// ---- DUTs/IO/Boxes/EL1808_78E8D3DD.TcDUT
{attribute 'GeneratedUsingTerminal: EL1808-0000-0016'}
{attribute addProperty BoxType "EL1808-0000-0016"}
{attribute addProperty Description "EL1808 8Ch. Dig. Input 24V, 3ms"}
{attribute addProperty Physics "KK"}
{attribute addProperty Id "Channel_1AT %I*Channel_830843C11Channel_2AT %I*Channel_830843C11Channel_3AT %I*Channel_830843C11Channel_4AT %I*Channel_830843C11Channel_5AT %I*Channel_830843C11Channel_6AT %I*Channel_830843C11Channel_7AT %I*Channel_830843C11Channel_8AT %I*Channel_830843C11WcStateAT %I*WcState_9091E0EB2InfoDataAT %I*InfoData_6F19DB2B2"}
{attribute addProperty CRC "2028524509"}
{attribute addProperty Size "12"}
TYPE EL1808_78E8D3DD EXTENDS EtcSlaveTerminalBase_947E5A46 :
STRUCT
	{attribute addProperty Name "Channel_1"}
	Channel_1 : Channel_830843C1;
	{attribute addProperty Name "Channel_2"}
	Channel_2 : Channel_830843C1;
	{attribute addProperty Name "Channel_3"}
	Channel_3 : Channel_830843C1;
	{attribute addProperty Name "Channel_4"}
	Channel_4 : Channel_830843C1;
	{attribute addProperty Name "Channel_5"}
	Channel_5 : Channel_830843C1;
	{attribute addProperty Name "Channel_6"}
	Channel_6 : Channel_830843C1;
	{attribute addProperty Name "Channel_7"}
	Channel_7 : Channel_830843C1;
	{attribute addProperty Name "Channel_8"}
	Channel_8 : Channel_830843C1;
	{attribute addProperty Name "WcState"}
	WcState : WcState_9091E0EB;
	{attribute addProperty Name "InfoData"}
	InfoData : InfoData_6F19DB2B;
END_STRUCT
END_TYPE

// ---- DUTs/IO/Boxes/EL1809_32157CFD.TcDUT
{attribute 'GeneratedUsingTerminal: EL1809-0000-0016'}
{attribute addProperty BoxType "EL1809-0000-0016"}
{attribute addProperty Description "EL1809 16Ch. Dig. Input 24V, 3ms"}
{attribute addProperty Physics "KK"}
{attribute addProperty Id "Channel_1AT %I*Channel_830843C11Channel_2AT %I*Channel_830843C11Channel_3AT %I*Channel_830843C11Channel_4AT %I*Channel_830843C11Channel_5AT %I*Channel_830843C11Channel_6AT %I*Channel_830843C11Channel_7AT %I*Channel_830843C11Channel_8AT %I*Channel_830843C11Channel_9AT %I*Channel_830843C11Channel_10AT %I*Channel_830843C11Channel_11AT %I*Channel_830843C11Channel_12AT %I*Channel_830843C11Channel_13AT %I*Channel_830843C11Channel_14AT %I*Channel_830843C11Channel_15AT %I*Channel_830843C11Channel_16AT %I*Channel_830843C11WcStateAT %I*WcState_9091E0EB2InfoDataAT %I*InfoData_6F19DB2B2"}
{attribute addProperty CRC "840269053"}
{attribute addProperty Size "20"}
TYPE EL1809_32157CFD EXTENDS EtcSlaveTerminalBase_947E5A46 :
STRUCT
	{attribute addProperty Name "Channel_1"}
	Channel_1 : Channel_830843C1;
	{attribute addProperty Name "Channel_2"}
	Channel_2 : Channel_830843C1;
	{attribute addProperty Name "Channel_3"}
	Channel_3 : Channel_830843C1;
	{attribute addProperty Name "Channel_4"}
	Channel_4 : Channel_830843C1;
	{attribute addProperty Name "Channel_5"}
	Channel_5 : Channel_830843C1;
	{attribute addProperty Name "Channel_6"}
	Channel_6 : Channel_830843C1;
	{attribute addProperty Name "Channel_7"}
	Channel_7 : Channel_830843C1;
	{attribute addProperty Name "Channel_8"}
	Channel_8 : Channel_830843C1;
	{attribute addProperty Name "Channel_9"}
	Channel_9 : Channel_830843C1;
	{attribute addProperty Name "Channel_10"}
	Channel_10 : Channel_830843C1;
	{attribute addProperty Name "Channel_11"}
	Channel_11 : Channel_830843C1;
	{attribute addProperty Name "Channel_12"}
	Channel_12 : Channel_830843C1;
	{attribute addProperty Name "Channel_13"}
	Channel_13 : Channel_830843C1;
	{attribute addProperty Name "Channel_14"}
	Channel_14 : Channel_830843C1;
	{attribute addProperty Name "Channel_15"}
	Channel_15 : Channel_830843C1;
	{attribute addProperty Name "Channel_16"}
	Channel_16 : Channel_830843C1;
	{attribute addProperty Name "WcState"}
	WcState : WcState_9091E0EB;
	{attribute addProperty Name "InfoData"}
	InfoData : InfoData_6F19DB2B;
END_STRUCT
END_TYPE

// ---- DUTs/IO/Boxes/EL1814_D135F8DB.TcDUT
{attribute 'GeneratedUsingTerminal: EL1814-0000-0016'}
{attribute addProperty BoxType "EL1814-0000-0016"}
{attribute addProperty Description "EL1814 4Ch. Dig. Input 24V, 10µs"}
{attribute addProperty Physics "KK"}
{attribute addProperty Id "Channel_1AT %I*Channel_830843C11Channel_2AT %I*Channel_830843C11Channel_3AT %I*Channel_830843C11Channel_4AT %I*Channel_830843C11WcStateAT %I*WcState_9091E0EB2InfoDataAT %I*InfoData_6F19DB2B2"}
{attribute addProperty CRC "3509975259"}
{attribute addProperty Size "8"}
TYPE EL1814_D135F8DB EXTENDS EtcSlaveTerminalBase_947E5A46 :
STRUCT
	{attribute addProperty Name "Channel_1"}
	Channel_1 : Channel_830843C1;
	{attribute addProperty Name "Channel_2"}
	Channel_2 : Channel_830843C1;
	{attribute addProperty Name "Channel_3"}
	Channel_3 : Channel_830843C1;
	{attribute addProperty Name "Channel_4"}
	Channel_4 : Channel_830843C1;
	{attribute addProperty Name "WcState"}
	WcState : WcState_9091E0EB;
	{attribute addProperty Name "InfoData"}
	InfoData : InfoData_6F19DB2B;
END_STRUCT
END_TYPE

// ---- DUTs/IO/Boxes/EL1819_32157CFD.TcDUT
{attribute 'GeneratedUsingTerminal: EL1819-0000-0016'}
{attribute addProperty BoxType "EL1819-0000-0016"}
{attribute addProperty Description "EL1819 16Ch. Dig. Input 24V, 10µs"}
{attribute addProperty Physics "KK"}
{attribute addProperty Id "Channel_1AT %I*Channel_830843C11Channel_2AT %I*Channel_830843C11Channel_3AT %I*Channel_830843C11Channel_4AT %I*Channel_830843C11Channel_5AT %I*Channel_830843C11Channel_6AT %I*Channel_830843C11Channel_7AT %I*Channel_830843C11Channel_8AT %I*Channel_830843C11Channel_9AT %I*Channel_830843C11Channel_10AT %I*Channel_830843C11Channel_11AT %I*Channel_830843C11Channel_12AT %I*Channel_830843C11Channel_13AT %I*Channel_830843C11Channel_14AT %I*Channel_830843C11Channel_15AT %I*Channel_830843C11Channel_16AT %I*Channel_830843C11WcStateAT %I*WcState_9091E0EB2InfoDataAT %I*InfoData_6F19DB2B2"}
{attribute addProperty CRC "840269053"}
{attribute addProperty Size "20"}
TYPE EL1819_32157CFD EXTENDS EtcSlaveTerminalBase_947E5A46 :
STRUCT
	{attribute addProperty Name "Channel_1"}
	Channel_1 : Channel_830843C1;
	{attribute addProperty Name "Channel_2"}
	Channel_2 : Channel_830843C1;
	{attribute addProperty Name "Channel_3"}
	Channel_3 : Channel_830843C1;
	{attribute addProperty Name "Channel_4"}
	Channel_4 : Channel_830843C1;
	{attribute addProperty Name "Channel_5"}
	Channel_5 : Channel_830843C1;
	{attribute addProperty Name "Channel_6"}
	Channel_6 : Channel_830843C1;
	{attribute addProperty Name "Channel_7"}
	Channel_7 : Channel_830843C1;
	{attribute addProperty Name "Channel_8"}
	Channel_8 : Channel_830843C1;
	{attribute addProperty Name "Channel_9"}
	Channel_9 : Channel_830843C1;
	{attribute addProperty Name "Channel_10"}
	Channel_10 : Channel_830843C1;
	{attribute addProperty Name "Channel_11"}
	Channel_11 : Channel_830843C1;
	{attribute addProperty Name "Channel_12"}
	Channel_12 : Channel_830843C1;
	{attribute addProperty Name "Channel_13"}
	Channel_13 : Channel_830843C1;
	{attribute addProperty Name "Channel_14"}
	Channel_14 : Channel_830843C1;
	{attribute addProperty Name "Channel_15"}
	Channel_15 : Channel_830843C1;
	{attribute addProperty Name "Channel_16"}
	Channel_16 : Channel_830843C1;
	{attribute addProperty Name "WcState"}
	WcState : WcState_9091E0EB;
	{attribute addProperty Name "InfoData"}
	InfoData : InfoData_6F19DB2B;
END_STRUCT
END_TYPE

// ---- DUTs/IO/Boxes/EL1852_7699BCF6.TcDUT
{attribute 'GeneratedUsingTerminal: EL1852-0000-0016'}
{attribute addProperty BoxType "EL1852-0000-0016"}
{attribute addProperty Description "EL1852 8Ch. Dig. Input 24V, 3ms, 8Ch. Dig. Output 24V, 0.5A"}
{attribute addProperty Physics "KK"}
{attribute addProperty Id "Channel_1AT %I*Channel_830843C11Channel_2AT %I*Channel_830843C11Channel_3AT %I*Channel_830843C11Channel_4AT %I*Channel_830843C11Channel_5AT %I*Channel_830843C11Channel_6AT %I*Channel_830843C11Channel_7AT %I*Channel_830843C11Channel_8AT %I*Channel_830843C11Channel_9AT %Q*Channel_42CA91F71Channel_10AT %Q*Channel_42CA91F71Channel_11AT %Q*Channel_42CA91F71Channel_12AT %Q*Channel_42CA91F71Channel_13AT %Q*Channel_42CA91F71Channel_14AT %Q*Channel_42CA91F71Channel_15AT %Q*Channel_42CA91F71Channel_16AT %Q*Channel_42CA91F71WcStateAT %I*WcState_9091E0EB2InfoDataAT %I*InfoData_6F19DB2B2"}
{attribute addProperty CRC "1989786870"}
{attribute addProperty Size "20"}
TYPE EL1852_7699BCF6 EXTENDS EtcSlaveTerminalBase_947E5A46 :
STRUCT
	{attribute addProperty Name "Channel_1"}
	Channel_1 : Channel_830843C1;
	{attribute addProperty Name "Channel_2"}
	Channel_2 : Channel_830843C1;
	{attribute addProperty Name "Channel_3"}
	Channel_3 : Channel_830843C1;
	{attribute addProperty Name "Channel_4"}
	Channel_4 : Channel_830843C1;
	{attribute addProperty Name "Channel_5"}
	Channel_5 : Channel_830843C1;
	{attribute addProperty Name "Channel_6"}
	Channel_6 : Channel_830843C1;
	{attribute addProperty Name "Channel_7"}
	Channel_7 : Channel_830843C1;
	{attribute addProperty Name "Channel_8"}
	Channel_8 : Channel_830843C1;
	{attribute addProperty Name "Channel_9"}
	Channel_9 : Channel_42CA91F7;
	{attribute addProperty Name "Channel_10"}
	Channel_10 : Channel_42CA91F7;
	{attribute addProperty Name "Channel_11"}
	Channel_11 : Channel_42CA91F7;
	{attribute addProperty Name "Channel_12"}
	Channel_12 : Channel_42CA91F7;
	{attribute addProperty Name "Channel_13"}
	Channel_13 : Channel_42CA91F7;
	{attribute addProperty Name "Channel_14"}
	Channel_14 : Channel_42CA91F7;
	{attribute addProperty Name "Channel_15"}
	Channel_15 : Channel_42CA91F7;
	{attribute addProperty Name "Channel_16"}
	Channel_16 : Channel_42CA91F7;
	{attribute addProperty Name "WcState"}
	WcState : WcState_9091E0EB;
	{attribute addProperty Name "InfoData"}
	InfoData : InfoData_6F19DB2B;
END_STRUCT
END_TYPE

// ---- DUTs/IO/Boxes/EL1859_7699BCF6.TcDUT
{attribute 'GeneratedUsingTerminal: EL1859-0000-0016'}
{attribute addProperty BoxType "EL1859-0000-0016"}
{attribute addProperty Description "EL1859 8Ch. Dig. Input 24V, 3ms, 8Ch. Dig. Output 24V, 0.5A"}
{attribute addProperty Physics "KK"}
{attribute addProperty Id "Channel_1AT %I*Channel_830843C11Channel_2AT %I*Channel_830843C11Channel_3AT %I*Channel_830843C11Channel_4AT %I*Channel_830843C11Channel_5AT %I*Channel_830843C11Channel_6AT %I*Channel_830843C11Channel_7AT %I*Channel_830843C11Channel_8AT %I*Channel_830843C11Channel_9AT %Q*Channel_42CA91F71Channel_10AT %Q*Channel_42CA91F71Channel_11AT %Q*Channel_42CA91F71Channel_12AT %Q*Channel_42CA91F71Channel_13AT %Q*Channel_42CA91F71Channel_14AT %Q*Channel_42CA91F71Channel_15AT %Q*Channel_42CA91F71Channel_16AT %Q*Channel_42CA91F71WcStateAT %I*WcState_9091E0EB2InfoDataAT %I*InfoData_6F19DB2B2"}
{attribute addProperty CRC "1989786870"}
{attribute addProperty Size "20"}
TYPE EL1859_7699BCF6 EXTENDS EtcSlaveTerminalBase_947E5A46 :
STRUCT
	{attribute addProperty Name "Channel_1"}
	Channel_1 : Channel_830843C1;
	{attribute addProperty Name "Channel_2"}
	Channel_2 : Channel_830843C1;
	{attribute addProperty Name "Channel_3"}
	Channel_3 : Channel_830843C1;
	{attribute addProperty Name "Channel_4"}
	Channel_4 : Channel_830843C1;
	{attribute addProperty Name "Channel_5"}
	Channel_5 : Channel_830843C1;
	{attribute addProperty Name "Channel_6"}
	Channel_6 : Channel_830843C1;
	{attribute addProperty Name "Channel_7"}
	Channel_7 : Channel_830843C1;
	{attribute addProperty Name "Channel_8"}
	Channel_8 : Channel_830843C1;
	{attribute addProperty Name "Channel_9"}
	Channel_9 : Channel_42CA91F7;
	{attribute addProperty Name "Channel_10"}
	Channel_10 : Channel_42CA91F7;
	{attribute addProperty Name "Channel_11"}
	Channel_11 : Channel_42CA91F7;
	{attribute addProperty Name "Channel_12"}
	Channel_12 : Channel_42CA91F7;
	{attribute addProperty Name "Channel_13"}
	Channel_13 : Channel_42CA91F7;
	{attribute addProperty Name "Channel_14"}
	Channel_14 : Channel_42CA91F7;
	{attribute addProperty Name "Channel_15"}
	Channel_15 : Channel_42CA91F7;
	{attribute addProperty Name "Channel_16"}
	Channel_16 : Channel_42CA91F7;
	{attribute addProperty Name "WcState"}
	WcState : WcState_9091E0EB;
	{attribute addProperty Name "InfoData"}
	InfoData : InfoData_6F19DB2B;
END_STRUCT
END_TYPE

// ---- DUTs/IO/Boxes/EL1862_32157CFD.TcDUT
{attribute 'GeneratedUsingTerminal: EL1862-0000-0016'}
{attribute addProperty BoxType "EL1862-0000-0016"}
{attribute addProperty Description "EL1862 16Ch. Dig. Input 24V, 3ms"}
{attribute addProperty Physics "KK"}
{attribute addProperty Id "Channel_1AT %I*Channel_830843C11Channel_2AT %I*Channel_830843C11Channel_3AT %I*Channel_830843C11Channel_4AT %I*Channel_830843C11Channel_5AT %I*Channel_830843C11Channel_6AT %I*Channel_830843C11Channel_7AT %I*Channel_830843C11Channel_8AT %I*Channel_830843C11Channel_9AT %I*Channel_830843C11Channel_10AT %I*Channel_830843C11Channel_11AT %I*Channel_830843C11Channel_12AT %I*Channel_830843C11Channel_13AT %I*Channel_830843C11Channel_14AT %I*Channel_830843C11Channel_15AT %I*Channel_830843C11Channel_16AT %I*Channel_830843C11WcStateAT %I*WcState_9091E0EB2InfoDataAT %I*InfoData_6F19DB2B2"}
{attribute addProperty CRC "840269053"}
{attribute addProperty Size "20"}
TYPE EL1862_32157CFD EXTENDS EtcSlaveTerminalBase_947E5A46 :
STRUCT
	{attribute addProperty Name "Channel_1"}
	Channel_1 : Channel_830843C1;
	{attribute addProperty Name "Channel_2"}
	Channel_2 : Channel_830843C1;
	{attribute addProperty Name "Channel_3"}
	Channel_3 : Channel_830843C1;
	{attribute addProperty Name "Channel_4"}
	Channel_4 : Channel_830843C1;
	{attribute addProperty Name "Channel_5"}
	Channel_5 : Channel_830843C1;
	{attribute addProperty Name "Channel_6"}
	Channel_6 : Channel_830843C1;
	{attribute addProperty Name "Channel_7"}
	Channel_7 : Channel_830843C1;
	{attribute addProperty Name "Channel_8"}
	Channel_8 : Channel_830843C1;
	{attribute addProperty Name "Channel_9"}
	Channel_9 : Channel_830843C1;
	{attribute addProperty Name "Channel_10"}
	Channel_10 : Channel_830843C1;
	{attribute addProperty Name "Channel_11"}
	Channel_11 : Channel_830843C1;
	{attribute addProperty Name "Channel_12"}
	Channel_12 : Channel_830843C1;
	{attribute addProperty Name "Channel_13"}
	Channel_13 : Channel_830843C1;
	{attribute addProperty Name "Channel_14"}
	Channel_14 : Channel_830843C1;
	{attribute addProperty Name "Channel_15"}
	Channel_15 : Channel_830843C1;
	{attribute addProperty Name "Channel_16"}
	Channel_16 : Channel_830843C1;
	{attribute addProperty Name "WcState"}
	WcState : WcState_9091E0EB;
	{attribute addProperty Name "InfoData"}
	InfoData : InfoData_6F19DB2B;
END_STRUCT
END_TYPE

// ---- DUTs/IO/Boxes/EL1872_32157CFD.TcDUT
{attribute 'GeneratedUsingTerminal: EL1872-0000-0016'}
{attribute addProperty BoxType "EL1872-0000-0016"}
{attribute addProperty Description "EL1872 16Ch. Dig. Input 24V, 10µs"}
{attribute addProperty Physics "KK"}
{attribute addProperty Id "Channel_1AT %I*Channel_830843C11Channel_2AT %I*Channel_830843C11Channel_3AT %I*Channel_830843C11Channel_4AT %I*Channel_830843C11Channel_5AT %I*Channel_830843C11Channel_6AT %I*Channel_830843C11Channel_7AT %I*Channel_830843C11Channel_8AT %I*Channel_830843C11Channel_9AT %I*Channel_830843C11Channel_10AT %I*Channel_830843C11Channel_11AT %I*Channel_830843C11Channel_12AT %I*Channel_830843C11Channel_13AT %I*Channel_830843C11Channel_14AT %I*Channel_830843C11Channel_15AT %I*Channel_830843C11Channel_16AT %I*Channel_830843C11WcStateAT %I*WcState_9091E0EB2InfoDataAT %I*InfoData_6F19DB2B2"}
{attribute addProperty CRC "840269053"}
{attribute addProperty Size "20"}
TYPE EL1872_32157CFD EXTENDS EtcSlaveTerminalBase_947E5A46 :
STRUCT
	{attribute addProperty Name "Channel_1"}
	Channel_1 : Channel_830843C1;
	{attribute addProperty Name "Channel_2"}
	Channel_2 : Channel_830843C1;
	{attribute addProperty Name "Channel_3"}
	Channel_3 : Channel_830843C1;
	{attribute addProperty Name "Channel_4"}
	Channel_4 : Channel_830843C1;
	{attribute addProperty Name "Channel_5"}
	Channel_5 : Channel_830843C1;
	{attribute addProperty Name "Channel_6"}
	Channel_6 : Channel_830843C1;
	{attribute addProperty Name "Channel_7"}
	Channel_7 : Channel_830843C1;
	{attribute addProperty Name "Channel_8"}
	Channel_8 : Channel_830843C1;
	{attribute addProperty Name "Channel_9"}
	Channel_9 : Channel_830843C1;
	{attribute addProperty Name "Channel_10"}
	Channel_10 : Channel_830843C1;
	{attribute addProperty Name "Channel_11"}
	Channel_11 : Channel_830843C1;
	{attribute addProperty Name "Channel_12"}
	Channel_12 : Channel_830843C1;
	{attribute addProperty Name "Channel_13"}
	Channel_13 : Channel_830843C1;
	{attribute addProperty Name "Channel_14"}
	Channel_14 : Channel_830843C1;
	{attribute addProperty Name "Channel_15"}
	Channel_15 : Channel_830843C1;
	{attribute addProperty Name "Channel_16"}
	Channel_16 : Channel_830843C1;
	{attribute addProperty Name "WcState"}
	WcState : WcState_9091E0EB;
	{attribute addProperty Name "InfoData"}
	InfoData : InfoData_6F19DB2B;
END_STRUCT
END_TYPE

// ---- DUTs/IO/Boxes/EL1889_32157CFD.TcDUT
{attribute 'GeneratedUsingTerminal: EL1889-0000-0016'}
{attribute addProperty BoxType "EL1889-0000-0016"}
{attribute addProperty Description "EL1889 16Ch. Dig. Input 24V, 3ms, negative"}
{attribute addProperty Physics "KK"}
{attribute addProperty Id "Channel_1AT %I*Channel_830843C11Channel_2AT %I*Channel_830843C11Channel_3AT %I*Channel_830843C11Channel_4AT %I*Channel_830843C11Channel_5AT %I*Channel_830843C11Channel_6AT %I*Channel_830843C11Channel_7AT %I*Channel_830843C11Channel_8AT %I*Channel_830843C11Channel_9AT %I*Channel_830843C11Channel_10AT %I*Channel_830843C11Channel_11AT %I*Channel_830843C11Channel_12AT %I*Channel_830843C11Channel_13AT %I*Channel_830843C11Channel_14AT %I*Channel_830843C11Channel_15AT %I*Channel_830843C11Channel_16AT %I*Channel_830843C11WcStateAT %I*WcState_9091E0EB2InfoDataAT %I*InfoData_6F19DB2B2"}
{attribute addProperty CRC "840269053"}
{attribute addProperty Size "20"}
TYPE EL1889_32157CFD EXTENDS EtcSlaveTerminalBase_947E5A46 :
STRUCT
	{attribute addProperty Name "Channel_1"}
	Channel_1 : Channel_830843C1;
	{attribute addProperty Name "Channel_2"}
	Channel_2 : Channel_830843C1;
	{attribute addProperty Name "Channel_3"}
	Channel_3 : Channel_830843C1;
	{attribute addProperty Name "Channel_4"}
	Channel_4 : Channel_830843C1;
	{attribute addProperty Name "Channel_5"}
	Channel_5 : Channel_830843C1;
	{attribute addProperty Name "Channel_6"}
	Channel_6 : Channel_830843C1;
	{attribute addProperty Name "Channel_7"}
	Channel_7 : Channel_830843C1;
	{attribute addProperty Name "Channel_8"}
	Channel_8 : Channel_830843C1;
	{attribute addProperty Name "Channel_9"}
	Channel_9 : Channel_830843C1;
	{attribute addProperty Name "Channel_10"}
	Channel_10 : Channel_830843C1;
	{attribute addProperty Name "Channel_11"}
	Channel_11 : Channel_830843C1;
	{attribute addProperty Name "Channel_12"}
	Channel_12 : Channel_830843C1;
	{attribute addProperty Name "Channel_13"}
	Channel_13 : Channel_830843C1;
	{attribute addProperty Name "Channel_14"}
	Channel_14 : Channel_830843C1;
	{attribute addProperty Name "Channel_15"}
	Channel_15 : Channel_830843C1;
	{attribute addProperty Name "Channel_16"}
	Channel_16 : Channel_830843C1;
	{attribute addProperty Name "WcState"}
	WcState : WcState_9091E0EB;
	{attribute addProperty Name "InfoData"}
	InfoData : InfoData_6F19DB2B;
END_STRUCT
END_TYPE

// ---- DUTs/IO/Boxes/EL1899_32157CFD.TcDUT
{attribute 'GeneratedUsingTerminal: EL1899-0000-0016'}
{attribute addProperty BoxType "EL1899-0000-0016"}
{attribute addProperty Description "EL1899 16Ch. Dig. Input 24V, 10µs, negative"}
{attribute addProperty Physics "KK"}
{attribute addProperty Id "Channel_1AT %I*Channel_830843C11Channel_2AT %I*Channel_830843C11Channel_3AT %I*Channel_830843C11Channel_4AT %I*Channel_830843C11Channel_5AT %I*Channel_830843C11Channel_6AT %I*Channel_830843C11Channel_7AT %I*Channel_830843C11Channel_8AT %I*Channel_830843C11Channel_9AT %I*Channel_830843C11Channel_10AT %I*Channel_830843C11Channel_11AT %I*Channel_830843C11Channel_12AT %I*Channel_830843C11Channel_13AT %I*Channel_830843C11Channel_14AT %I*Channel_830843C11Channel_15AT %I*Channel_830843C11Channel_16AT %I*Channel_830843C11WcStateAT %I*WcState_9091E0EB2InfoDataAT %I*InfoData_6F19DB2B2"}
{attribute addProperty CRC "840269053"}
{attribute addProperty Size "20"}
TYPE EL1899_32157CFD EXTENDS EtcSlaveTerminalBase_947E5A46 :
STRUCT
	{attribute addProperty Name "Channel_1"}
	Channel_1 : Channel_830843C1;
	{attribute addProperty Name "Channel_2"}
	Channel_2 : Channel_830843C1;
	{attribute addProperty Name "Channel_3"}
	Channel_3 : Channel_830843C1;
	{attribute addProperty Name "Channel_4"}
	Channel_4 : Channel_830843C1;
	{attribute addProperty Name "Channel_5"}
	Channel_5 : Channel_830843C1;
	{attribute addProperty Name "Channel_6"}
	Channel_6 : Channel_830843C1;
	{attribute addProperty Name "Channel_7"}
	Channel_7 : Channel_830843C1;
	{attribute addProperty Name "Channel_8"}
	Channel_8 : Channel_830843C1;
	{attribute addProperty Name "Channel_9"}
	Channel_9 : Channel_830843C1;
	{attribute addProperty Name "Channel_10"}
	Channel_10 : Channel_830843C1;
	{attribute addProperty Name "Channel_11"}
	Channel_11 : Channel_830843C1;
	{attribute addProperty Name "Channel_12"}
	Channel_12 : Channel_830843C1;
	{attribute addProperty Name "Channel_13"}
	Channel_13 : Channel_830843C1;
	{attribute addProperty Name "Channel_14"}
	Channel_14 : Channel_830843C1;
	{attribute addProperty Name "Channel_15"}
	Channel_15 : Channel_830843C1;
	{attribute addProperty Name "Channel_16"}
	Channel_16 : Channel_830843C1;
	{attribute addProperty Name "WcState"}
	WcState : WcState_9091E0EB;
	{attribute addProperty Name "InfoData"}
	InfoData : InfoData_6F19DB2B;
END_STRUCT
END_TYPE

// ---- DUTs/IO/Boxes/EL2002_B0214940.TcDUT
{attribute 'GeneratedUsingTerminal: EL2002--0000'}
{attribute addProperty BoxType "EL2002--0000"}
{attribute addProperty Description "EL2002 2Ch. Dig. Output 24V, 0.5A"}
{attribute addProperty Physics "KK"}
{attribute addProperty Id "Channel_1AT %Q*Channel_42CA91F71Channel_2AT %Q*Channel_42CA91F71WcStateAT %I*WcState_0B2B16F91InfoDataAT %I*InfoData_6F19DB2B2"}
{attribute addProperty CRC "2954971456"}
{attribute addProperty Size "5"}
TYPE EL2002_B0214940 EXTENDS EtcSlaveTerminalBase_947E5A46 :
STRUCT
	{attribute addProperty Name "Channel_1"}
	Channel_1 : Channel_42CA91F7;
	{attribute addProperty Name "Channel_2"}
	Channel_2 : Channel_42CA91F7;
	{attribute addProperty Name "WcState"}
	WcState : WcState_0B2B16F9;
	{attribute addProperty Name "InfoData"}
	InfoData : InfoData_6F19DB2B;
END_STRUCT
END_TYPE

// ---- DUTs/IO/Boxes/EL2004_7B64371E.TcDUT
{attribute 'GeneratedUsingTerminal: EL2004--0000'}
{attribute addProperty BoxType "EL2004--0000"}
{attribute addProperty Description "EL2004 4Ch. Dig. Output 24V, 0.5A"}
{attribute addProperty Physics "KK"}
{attribute addProperty Id "Channel_1AT %Q*Channel_42CA91F71Channel_2AT %Q*Channel_42CA91F71Channel_3AT %Q*Channel_42CA91F71Channel_4AT %Q*Channel_42CA91F71WcStateAT %I*WcState_0B2B16F91InfoDataAT %I*InfoData_6F19DB2B2"}
{attribute addProperty CRC "2070165278"}
{attribute addProperty Size "7"}
TYPE EL2004_7B64371E EXTENDS EtcSlaveTerminalBase_947E5A46 :
STRUCT
	{attribute addProperty Name "Channel_1"}
	Channel_1 : Channel_42CA91F7;
	{attribute addProperty Name "Channel_2"}
	Channel_2 : Channel_42CA91F7;
	{attribute addProperty Name "Channel_3"}
	Channel_3 : Channel_42CA91F7;
	{attribute addProperty Name "Channel_4"}
	Channel_4 : Channel_42CA91F7;
	{attribute addProperty Name "WcState"}
	WcState : WcState_0B2B16F9;
	{attribute addProperty Name "InfoData"}
	InfoData : InfoData_6F19DB2B;
END_STRUCT
END_TYPE

// ---- DUTs/IO/Boxes/EL2008_E2806B95.TcDUT
{attribute 'GeneratedUsingTerminal: EL2008-0000-0016'}
{attribute addProperty BoxType "EL2008-0000-0016"}
{attribute addProperty Description "EL2008 8Ch. Dig. Output 24V, 0.5A"}
{attribute addProperty Physics "KK"}
{attribute addProperty Id "Channel_1AT %Q*Channel_42CA91F71Channel_2AT %Q*Channel_42CA91F71Channel_3AT %Q*Channel_42CA91F71Channel_4AT %Q*Channel_42CA91F71Channel_5AT %Q*Channel_42CA91F71Channel_6AT %Q*Channel_42CA91F71Channel_7AT %Q*Channel_42CA91F71Channel_8AT %Q*Channel_42CA91F71WcStateAT %I*WcState_0B2B16F91InfoDataAT %I*InfoData_6F19DB2B2"}
{attribute addProperty CRC "3800066965"}
{attribute addProperty Size "11"}
TYPE EL2008_E2806B95 EXTENDS EtcSlaveTerminalBase_947E5A46 :
STRUCT
	{attribute addProperty Name "Channel_1"}
	Channel_1 : Channel_42CA91F7;
	{attribute addProperty Name "Channel_2"}
	Channel_2 : Channel_42CA91F7;
	{attribute addProperty Name "Channel_3"}
	Channel_3 : Channel_42CA91F7;
	{attribute addProperty Name "Channel_4"}
	Channel_4 : Channel_42CA91F7;
	{attribute addProperty Name "Channel_5"}
	Channel_5 : Channel_42CA91F7;
	{attribute addProperty Name "Channel_6"}
	Channel_6 : Channel_42CA91F7;
	{attribute addProperty Name "Channel_7"}
	Channel_7 : Channel_42CA91F7;
	{attribute addProperty Name "Channel_8"}
	Channel_8 : Channel_42CA91F7;
	{attribute addProperty Name "WcState"}
	WcState : WcState_0B2B16F9;
	{attribute addProperty Name "InfoData"}
	InfoData : InfoData_6F19DB2B;
END_STRUCT
END_TYPE

// ---- DUTs/IO/Boxes/EL2014_12F3E4E3.TcDUT
{attribute 'GeneratedUsingTerminal: EL2014-0000-0016'}
{attribute addProperty BoxType "EL2014-0000-0016"}
{attribute addProperty Description "EL2014 4Ch. Dig. Output 24V, 0,5A, Diagnostic"}
{attribute addProperty Physics "KK"}
{attribute addProperty Id "DIG_Diag_InputsAT %I*DIG_Diag_Inputs_58F3E2A816DIG_Inputs_DeviceAT %I*DIG_Inputs_Device_A1F150A94DIG_OutputsAT %Q*DIG_Outputs_F9744C664WcStateAT %I*WcState_9091E0EB2InfoDataAT %I*InfoData_32EB74EA10"}
{attribute addProperty CRC "317973731"}
{attribute addProperty Size "36"}
TYPE EL2014_12F3E4E3 EXTENDS EtcSlaveTerminalBase_947E5A46 :
STRUCT
	{attribute addProperty Name "DIG_Diag_Inputs"}
	DIG_Diag_Inputs : DIG_Diag_Inputs_58F3E2A8;
	{attribute addProperty Name "DIG_Inputs_Device"}
	DIG_Inputs_Device : DIG_Inputs_Device_A1F150A9;
	{attribute addProperty Name "DIG_Outputs"}
	DIG_Outputs : DIG_Outputs_F9744C66;
	{attribute addProperty Name "WcState"}
	WcState : WcState_9091E0EB;
	{attribute addProperty Name "InfoData"}
	InfoData : InfoData_32EB74EA;
END_STRUCT
END_TYPE

// ---- DUTs/IO/Boxes/EL2022_B0214940.TcDUT
{attribute 'GeneratedUsingTerminal: EL2022-0000-0016'}
{attribute addProperty BoxType "EL2022-0000-0016"}
{attribute addProperty Description "EL2022 2Ch. Dig. Output 24V, 2A"}
{attribute addProperty Physics "KK"}
{attribute addProperty Id "Channel_1AT %Q*Channel_42CA91F71Channel_2AT %Q*Channel_42CA91F71WcStateAT %I*WcState_0B2B16F91InfoDataAT %I*InfoData_6F19DB2B2"}
{attribute addProperty CRC "2954971456"}
{attribute addProperty Size "5"}
TYPE EL2022_B0214940 EXTENDS EtcSlaveTerminalBase_947E5A46 :
STRUCT
	{attribute addProperty Name "Channel_1"}
	Channel_1 : Channel_42CA91F7;
	{attribute addProperty Name "Channel_2"}
	Channel_2 : Channel_42CA91F7;
	{attribute addProperty Name "WcState"}
	WcState : WcState_0B2B16F9;
	{attribute addProperty Name "InfoData"}
	InfoData : InfoData_6F19DB2B;
END_STRUCT
END_TYPE

// ---- DUTs/IO/Boxes/EL2024_7B64371E.TcDUT
{attribute 'GeneratedUsingTerminal: EL2024-0000-0016'}
{attribute addProperty BoxType "EL2024-0000-0016"}
{attribute addProperty Description "EL2024 4Ch. Dig. Output 24V, 2A"}
{attribute addProperty Physics "KK"}
{attribute addProperty Id "Channel_1AT %Q*Channel_42CA91F71Channel_2AT %Q*Channel_42CA91F71Channel_3AT %Q*Channel_42CA91F71Channel_4AT %Q*Channel_42CA91F71WcStateAT %I*WcState_0B2B16F91InfoDataAT %I*InfoData_6F19DB2B2"}
{attribute addProperty CRC "2070165278"}
{attribute addProperty Size "7"}
TYPE EL2024_7B64371E EXTENDS EtcSlaveTerminalBase_947E5A46 :
STRUCT
	{attribute addProperty Name "Channel_1"}
	Channel_1 : Channel_42CA91F7;
	{attribute addProperty Name "Channel_2"}
	Channel_2 : Channel_42CA91F7;
	{attribute addProperty Name "Channel_3"}
	Channel_3 : Channel_42CA91F7;
	{attribute addProperty Name "Channel_4"}
	Channel_4 : Channel_42CA91F7;
	{attribute addProperty Name "WcState"}
	WcState : WcState_0B2B16F9;
	{attribute addProperty Name "InfoData"}
	InfoData : InfoData_6F19DB2B;
END_STRUCT
END_TYPE

// ---- DUTs/IO/Boxes/EL2032_4C3AB2A4.TcDUT
{attribute 'GeneratedUsingTerminal: EL2032--0000'}
{attribute addProperty BoxType "EL2032--0000"}
{attribute addProperty Description "EL2032 2Ch. Dig. Output 24V, 2A Diag"}
{attribute addProperty Physics "KK"}
{attribute addProperty Id "Diag_1AT %I*Diag_A72B1E171Diag_2AT %I*Diag_A72B1E171Channel_1AT %Q*Channel_42CA91F71Channel_2AT %Q*Channel_42CA91F71WcStateAT %I*WcState_9091E0EB2InfoDataAT %I*InfoData_6F19DB2B2"}
{attribute addProperty CRC "1278915236"}
{attribute addProperty Size "8"}
TYPE EL2032_4C3AB2A4 EXTENDS EtcSlaveTerminalBase_947E5A46 :
STRUCT
	{attribute addProperty Name "Diag_1"}
	Diag_1 : Diag_A72B1E17;
	{attribute addProperty Name "Diag_2"}
	Diag_2 : Diag_A72B1E17;
	{attribute addProperty Name "Channel_1"}
	Channel_1 : Channel_42CA91F7;
	{attribute addProperty Name "Channel_2"}
	Channel_2 : Channel_42CA91F7;
	{attribute addProperty Name "WcState"}
	WcState : WcState_9091E0EB;
	{attribute addProperty Name "InfoData"}
	InfoData : InfoData_6F19DB2B;
END_STRUCT
END_TYPE

// ---- DUTs/IO/Boxes/EL2034_9227BD07.TcDUT
{attribute 'GeneratedUsingTerminal: EL2034-0000-0016'}
{attribute addProperty BoxType "EL2034-0000-0016"}
{attribute addProperty Description "EL2034 4Ch. Dig. Output 24V, 2A, Diagnostic"}
{attribute addProperty Physics "KK"}
{attribute addProperty Id "Diag_1AT %I*Diag_A72B1E171Diag_2AT %I*Diag_A72B1E171Diag_3AT %I*Diag_A72B1E171Diag_4AT %I*Diag_A72B1E171Channel_1AT %Q*Channel_42CA91F71Channel_2AT %Q*Channel_42CA91F71Channel_3AT %Q*Channel_42CA91F71Channel_4AT %Q*Channel_42CA91F71WcStateAT %I*WcState_9091E0EB2InfoDataAT %I*InfoData_6F19DB2B2"}
{attribute addProperty CRC "2452077831"}
{attribute addProperty Size "12"}
TYPE EL2034_9227BD07 EXTENDS EtcSlaveTerminalBase_947E5A46 :
STRUCT
	{attribute addProperty Name "Diag_1"}
	Diag_1 : Diag_A72B1E17;
	{attribute addProperty Name "Diag_2"}
	Diag_2 : Diag_A72B1E17;
	{attribute addProperty Name "Diag_3"}
	Diag_3 : Diag_A72B1E17;
	{attribute addProperty Name "Diag_4"}
	Diag_4 : Diag_A72B1E17;
	{attribute addProperty Name "Channel_1"}
	Channel_1 : Channel_42CA91F7;
	{attribute addProperty Name "Channel_2"}
	Channel_2 : Channel_42CA91F7;
	{attribute addProperty Name "Channel_3"}
	Channel_3 : Channel_42CA91F7;
	{attribute addProperty Name "Channel_4"}
	Channel_4 : Channel_42CA91F7;
	{attribute addProperty Name "WcState"}
	WcState : WcState_9091E0EB;
	{attribute addProperty Name "InfoData"}
	InfoData : InfoData_6F19DB2B;
END_STRUCT
END_TYPE

// ---- DUTs/IO/Boxes/EL2042_B0214940.TcDUT
{attribute 'GeneratedUsingTerminal: EL2042-0000-0016'}
{attribute addProperty BoxType "EL2042-0000-0016"}
{attribute addProperty Description "EL2042 2Ch. Dig. Output 24V, 4A"}
{attribute addProperty Physics "KK"}
{attribute addProperty Id "Channel_1AT %Q*Channel_42CA91F71Channel_2AT %Q*Channel_42CA91F71WcStateAT %I*WcState_0B2B16F91InfoDataAT %I*InfoData_6F19DB2B2"}
{attribute addProperty CRC "2954971456"}
{attribute addProperty Size "5"}
TYPE EL2042_B0214940 EXTENDS EtcSlaveTerminalBase_947E5A46 :
STRUCT
	{attribute addProperty Name "Channel_1"}
	Channel_1 : Channel_42CA91F7;
	{attribute addProperty Name "Channel_2"}
	Channel_2 : Channel_42CA91F7;
	{attribute addProperty Name "WcState"}
	WcState : WcState_0B2B16F9;
	{attribute addProperty Name "InfoData"}
	InfoData : InfoData_6F19DB2B;
END_STRUCT
END_TYPE

// ---- DUTs/IO/Boxes/EL2044_12F3E4E3.TcDUT
{attribute 'GeneratedUsingTerminal: EL2044-0000-0016'}
{attribute addProperty BoxType "EL2044-0000-0016"}
{attribute addProperty Description "EL2044 4Ch. Dig. Output 24V, 2A, Diagnostic"}
{attribute addProperty Physics "KK"}
{attribute addProperty Id "DIG_Diag_InputsAT %I*DIG_Diag_Inputs_58F3E2A816DIG_Inputs_DeviceAT %I*DIG_Inputs_Device_A1F150A94DIG_OutputsAT %Q*DIG_Outputs_F9744C664WcStateAT %I*WcState_9091E0EB2InfoDataAT %I*InfoData_32EB74EA10"}
{attribute addProperty CRC "317973731"}
{attribute addProperty Size "36"}
TYPE EL2044_12F3E4E3 EXTENDS EtcSlaveTerminalBase_947E5A46 :
STRUCT
	{attribute addProperty Name "DIG_Diag_Inputs"}
	DIG_Diag_Inputs : DIG_Diag_Inputs_58F3E2A8;
	{attribute addProperty Name "DIG_Inputs_Device"}
	DIG_Inputs_Device : DIG_Inputs_Device_A1F150A9;
	{attribute addProperty Name "DIG_Outputs"}
	DIG_Outputs : DIG_Outputs_F9744C66;
	{attribute addProperty Name "WcState"}
	WcState : WcState_9091E0EB;
	{attribute addProperty Name "InfoData"}
	InfoData : InfoData_32EB74EA;
END_STRUCT
END_TYPE

// ---- DUTs/IO/Boxes/EL2084_7B64371E.TcDUT
{attribute 'GeneratedUsingTerminal: EL2084-0000-0016'}
{attribute addProperty BoxType "EL2084-0000-0016"}
{attribute addProperty Description "EL2084 4Ch. Dig. Output 24V, 0.5A, switching to negative"}
{attribute addProperty Physics "KK"}
{attribute addProperty Id "Channel_1AT %Q*Channel_42CA91F71Channel_2AT %Q*Channel_42CA91F71Channel_3AT %Q*Channel_42CA91F71Channel_4AT %Q*Channel_42CA91F71WcStateAT %I*WcState_0B2B16F91InfoDataAT %I*InfoData_6F19DB2B2"}
{attribute addProperty CRC "2070165278"}
{attribute addProperty Size "7"}
TYPE EL2084_7B64371E EXTENDS EtcSlaveTerminalBase_947E5A46 :
STRUCT
	{attribute addProperty Name "Channel_1"}
	Channel_1 : Channel_42CA91F7;
	{attribute addProperty Name "Channel_2"}
	Channel_2 : Channel_42CA91F7;
	{attribute addProperty Name "Channel_3"}
	Channel_3 : Channel_42CA91F7;
	{attribute addProperty Name "Channel_4"}
	Channel_4 : Channel_42CA91F7;
	{attribute addProperty Name "WcState"}
	WcState : WcState_0B2B16F9;
	{attribute addProperty Name "InfoData"}
	InfoData : InfoData_6F19DB2B;
END_STRUCT
END_TYPE

// ---- DUTs/IO/Boxes/EL2088_E2806B95.TcDUT
{attribute 'GeneratedUsingTerminal: EL2088-0000-0016'}
{attribute addProperty BoxType "EL2088-0000-0016"}
{attribute addProperty Description "EL2088 8Ch. Dig. Output 24V, 0.5A, switching to negative"}
{attribute addProperty Physics "KK"}
{attribute addProperty Id "Channel_1AT %Q*Channel_42CA91F71Channel_2AT %Q*Channel_42CA91F71Channel_3AT %Q*Channel_42CA91F71Channel_4AT %Q*Channel_42CA91F71Channel_5AT %Q*Channel_42CA91F71Channel_6AT %Q*Channel_42CA91F71Channel_7AT %Q*Channel_42CA91F71Channel_8AT %Q*Channel_42CA91F71WcStateAT %I*WcState_0B2B16F91InfoDataAT %I*InfoData_6F19DB2B2"}
{attribute addProperty CRC "3800066965"}
{attribute addProperty Size "11"}
TYPE EL2088_E2806B95 EXTENDS EtcSlaveTerminalBase_947E5A46 :
STRUCT
	{attribute addProperty Name "Channel_1"}
	Channel_1 : Channel_42CA91F7;
	{attribute addProperty Name "Channel_2"}
	Channel_2 : Channel_42CA91F7;
	{attribute addProperty Name "Channel_3"}
	Channel_3 : Channel_42CA91F7;
	{attribute addProperty Name "Channel_4"}
	Channel_4 : Channel_42CA91F7;
	{attribute addProperty Name "Channel_5"}
	Channel_5 : Channel_42CA91F7;
	{attribute addProperty Name "Channel_6"}
	Channel_6 : Channel_42CA91F7;
	{attribute addProperty Name "Channel_7"}
	Channel_7 : Channel_42CA91F7;
	{attribute addProperty Name "Channel_8"}
	Channel_8 : Channel_42CA91F7;
	{attribute addProperty Name "WcState"}
	WcState : WcState_0B2B16F9;
	{attribute addProperty Name "InfoData"}
	InfoData : InfoData_6F19DB2B;
END_STRUCT
END_TYPE

// ---- DUTs/IO/Boxes/EL2124_7B64371E.TcDUT
{attribute 'GeneratedUsingTerminal: EL2124-0000-0016'}
{attribute addProperty BoxType "EL2124-0000-0016"}
{attribute addProperty Description "EL2124 4Ch. Dig. Output 5V, 20mA"}
{attribute addProperty Physics "KK"}
{attribute addProperty Id "Channel_1AT %Q*Channel_42CA91F71Channel_2AT %Q*Channel_42CA91F71Channel_3AT %Q*Channel_42CA91F71Channel_4AT %Q*Channel_42CA91F71WcStateAT %I*WcState_0B2B16F91InfoDataAT %I*InfoData_6F19DB2B2"}
{attribute addProperty CRC "2070165278"}
{attribute addProperty Size "7"}
TYPE EL2124_7B64371E EXTENDS EtcSlaveTerminalBase_947E5A46 :
STRUCT
	{attribute addProperty Name "Channel_1"}
	Channel_1 : Channel_42CA91F7;
	{attribute addProperty Name "Channel_2"}
	Channel_2 : Channel_42CA91F7;
	{attribute addProperty Name "Channel_3"}
	Channel_3 : Channel_42CA91F7;
	{attribute addProperty Name "Channel_4"}
	Channel_4 : Channel_42CA91F7;
	{attribute addProperty Name "WcState"}
	WcState : WcState_0B2B16F9;
	{attribute addProperty Name "InfoData"}
	InfoData : InfoData_6F19DB2B;
END_STRUCT
END_TYPE

// ---- DUTs/IO/Boxes/EL2202_B0214940.TcDUT
{attribute 'GeneratedUsingTerminal: EL2202--0000'}
{attribute addProperty BoxType "EL2202--0000"}
{attribute addProperty Description "EL2202 2Ch. Dig. Output 24V, 0.5A, DC Sync"}
{attribute addProperty Physics "KK"}
{attribute addProperty Id "Channel_1AT %Q*Channel_42CA91F71Channel_2AT %Q*Channel_42CA91F71WcStateAT %I*WcState_0B2B16F91InfoDataAT %I*InfoData_6F19DB2B2"}
{attribute addProperty CRC "2954971456"}
{attribute addProperty Size "5"}
TYPE EL2202_B0214940 EXTENDS EtcSlaveTerminalBase_947E5A46 :
STRUCT
	{attribute addProperty Name "Channel_1"}
	Channel_1 : Channel_42CA91F7;
	{attribute addProperty Name "Channel_2"}
	Channel_2 : Channel_42CA91F7;
	{attribute addProperty Name "WcState"}
	WcState : WcState_0B2B16F9;
	{attribute addProperty Name "InfoData"}
	InfoData : InfoData_6F19DB2B;
END_STRUCT
END_TYPE

// ---- DUTs/IO/Boxes/EL2202_E4D0F256.TcDUT
{attribute 'GeneratedUsingTerminal: EL2202-0000-0016'}
{attribute addProperty BoxType "EL2202-0000-0016"}
{attribute addProperty Description "EL2202 2Ch. Dig. Output 24V, 0.5A"}
{attribute addProperty Physics "KK"}
{attribute addProperty Id "Channel_1AT %Q*Channel_54BE63B32Channel_2AT %Q*Channel_54BE63B32WcStateAT %I*WcState_0B2B16F91InfoDataAT %I*InfoData_6F19DB2B2"}
{attribute addProperty CRC "3838898774"}
{attribute addProperty Size "7"}
TYPE EL2202_E4D0F256 EXTENDS EtcSlaveTerminalBase_947E5A46 :
STRUCT
	{attribute addProperty Name "Channel_1"}
	Channel_1 : Channel_54BE63B3;
	{attribute addProperty Name "Channel_2"}
	Channel_2 : Channel_54BE63B3;
	{attribute addProperty Name "WcState"}
	WcState : WcState_0B2B16F9;
	{attribute addProperty Name "InfoData"}
	InfoData : InfoData_6F19DB2B;
END_STRUCT
END_TYPE

// ---- DUTs/IO/Boxes/EL2202_FB12F0C6.TcDUT
{attribute 'GeneratedUsingTerminal: EL2202-0100-0016'}
{attribute addProperty BoxType "EL2202-0100-0016"}
{attribute addProperty Description "EL2202-0100 2Ch. Dig. Output 24V, 0.5A, DC Sync"}
{attribute addProperty Physics "KK"}
{attribute addProperty Id "Channel_1AT %Q*Channel_54BE63B32Channel_2AT %Q*Channel_54BE63B32WcStateAT %I*WcState_0B2B16F91InfoDataAT %I*InfoData_A7436BC610"}
{attribute addProperty CRC "4212322502"}
{attribute addProperty Size "15"}
TYPE EL2202_FB12F0C6 EXTENDS EtcSlaveTerminalBase_947E5A46 :
STRUCT
	{attribute addProperty Name "Channel_1"}
	Channel_1 : Channel_54BE63B3;
	{attribute addProperty Name "Channel_2"}
	Channel_2 : Channel_54BE63B3;
	{attribute addProperty Name "WcState"}
	WcState : WcState_0B2B16F9;
	{attribute addProperty Name "InfoData"}
	InfoData : InfoData_A7436BC6;
END_STRUCT
END_TYPE

// ---- DUTs/IO/Boxes/EL2212_25BC0E0A.TcDUT
{attribute 'GeneratedUsingTerminal: EL2212-0000-0018'}
{attribute addProperty BoxType "EL2212-0000-0018"}
{attribute addProperty Description "EL2212 2Ch. dig. output with overexcitation (24V DC, 2.5A, 10A Peak)"}
{attribute addProperty Physics "KK"}
{attribute addProperty Id "DOX_Status_Channel_1AT %I*DOX_Status_Channel_09DD45C87DOX_Status_Channel_2AT %I*DOX_Status_Channel_09DD45C87DOX_Control_Channel_1AT %Q*DOX_Control_Channel_A74F23633DOX_Control_Channel_2AT %Q*DOX_Control_Channel_A74F23633WcStateAT %I*WcState_9091E0EB2InfoDataAT %I*InfoData_32EB74EA10"}
{attribute addProperty CRC "633081354"}
{attribute addProperty Size "32"}
TYPE EL2212_25BC0E0A EXTENDS EtcSlaveTerminalBase_947E5A46 :
STRUCT
	{attribute addProperty Name "DOX_Status_Channel_1"}
	DOX_Status_Channel_1 : DOX_Status_Channel_09DD45C8;
	{attribute addProperty Name "DOX_Status_Channel_2"}
	DOX_Status_Channel_2 : DOX_Status_Channel_09DD45C8;
	{attribute addProperty Name "DOX_Control_Channel_1"}
	DOX_Control_Channel_1 : DOX_Control_Channel_A74F2363;
	{attribute addProperty Name "DOX_Control_Channel_2"}
	DOX_Control_Channel_2 : DOX_Control_Channel_A74F2363;
	{attribute addProperty Name "WcState"}
	WcState : WcState_9091E0EB;
	{attribute addProperty Name "InfoData"}
	InfoData : InfoData_32EB74EA;
END_STRUCT
END_TYPE

// ---- DUTs/IO/Boxes/EL2212_C6DE6766.TcDUT
{attribute 'GeneratedUsingTerminal: EL2212-0000-0020'}
{attribute addProperty BoxType "EL2212-0000-0020"}
{attribute addProperty Description "EL2212 2Ch. dig. output with overexcitation (24V DC, 2.5A, 10A Peak)"}
{attribute addProperty Physics "KK"}
{attribute addProperty Id "DOX_Status_Channel_1AT %I*DOX_Status_Channel_6FDDBA987DOX_Status_Channel_2AT %I*DOX_Status_Channel_6FDDBA987DOX_Control_Channel_1AT %Q*DOX_Control_Channel_E69306414DOX_Control_Channel_2AT %Q*DOX_Control_Channel_E69306414WcStateAT %I*WcState_9091E0EB2InfoDataAT %I*InfoData_32EB74EA10"}
{attribute addProperty CRC "3336464230"}
{attribute addProperty Size "34"}
TYPE EL2212_C6DE6766 EXTENDS EtcSlaveTerminalBase_947E5A46 :
STRUCT
	{attribute addProperty Name "DOX_Status_Channel_1"}
	DOX_Status_Channel_1 : DOX_Status_Channel_6FDDBA98;
	{attribute addProperty Name "DOX_Status_Channel_2"}
	DOX_Status_Channel_2 : DOX_Status_Channel_6FDDBA98;
	{attribute addProperty Name "DOX_Control_Channel_1"}
	DOX_Control_Channel_1 : DOX_Control_Channel_E6930641;
	{attribute addProperty Name "DOX_Control_Channel_2"}
	DOX_Control_Channel_2 : DOX_Control_Channel_E6930641;
	{attribute addProperty Name "WcState"}
	WcState : WcState_9091E0EB;
	{attribute addProperty Name "InfoData"}
	InfoData : InfoData_32EB74EA;
END_STRUCT
END_TYPE

// ---- DUTs/IO/Boxes/EL2252_FF939DB0.TcDUT
{attribute 'GeneratedUsingTerminal: EL2252--0000'}
{attribute addProperty BoxType "EL2252--0000"}
{attribute addProperty Description "EL2252 2Ch. Dig. Output 24V, 0.5A, DC Time Stamp"}
{attribute addProperty Physics "KK"}
{attribute addProperty Id "DC_Sync_ActivateAT %Q*DC_Sync_Activate_FA2D29101DC_Sync_StartAT %Q*DC_Sync_Start_9CCB0E514Channel_1AT %Q*Channel_42CA91F71Channel_2AT %Q*Channel_42CA91F71WcStateAT %I*WcState_0B2B16F91InfoDataAT %I*InfoData_A7436BC610"}
{attribute addProperty CRC "4287864240"}
{attribute addProperty Size "18"}
TYPE EL2252_FF939DB0 EXTENDS EtcSlaveTerminalBase_947E5A46 :
STRUCT
	{attribute addProperty Name "DC_Sync_Activate"}
	DC_Sync_Activate : DC_Sync_Activate_FA2D2910;
	{attribute addProperty Name "DC_Sync_Start"}
	DC_Sync_Start : DC_Sync_Start_9CCB0E51;
	{attribute addProperty Name "Channel_1"}
	Channel_1 : Channel_42CA91F7;
	{attribute addProperty Name "Channel_2"}
	Channel_2 : Channel_42CA91F7;
	{attribute addProperty Name "WcState"}
	WcState : WcState_0B2B16F9;
	{attribute addProperty Name "InfoData"}
	InfoData : InfoData_A7436BC6;
END_STRUCT
END_TYPE

// ---- DUTs/IO/Boxes/EL2252_BD1134C6.TcDUT
{attribute 'GeneratedUsingTerminal: EL2252-0000-0016'}
{attribute addProperty BoxType "EL2252-0000-0016"}
{attribute addProperty Description "EL2252 2Ch. Dig. Output 24V, 0.5A, DC Time Stamp"}
{attribute addProperty Physics "KK"}
{attribute addProperty Id "DC_Sync_ActivateAT %Q*DC_Sync_Activate_FA2D29101DC_Sync_StartAT %Q*DC_Sync_Start_E82E92338Channel_1AT %Q*Channel_42CA91F71Channel_2AT %Q*Channel_42CA91F71WcStateAT %I*WcState_0B2B16F91InfoDataAT %I*InfoData_A7436BC610"}
{attribute addProperty CRC "3172021446"}
{attribute addProperty Size "22"}
TYPE EL2252_BD1134C6 EXTENDS EtcSlaveTerminalBase_947E5A46 :
STRUCT
	{attribute addProperty Name "DC_Sync_Activate"}
	DC_Sync_Activate : DC_Sync_Activate_FA2D2910;
	{attribute addProperty Name "DC_Sync_Start"}
	DC_Sync_Start : DC_Sync_Start_E82E9233;
	{attribute addProperty Name "Channel_1"}
	Channel_1 : Channel_42CA91F7;
	{attribute addProperty Name "Channel_2"}
	Channel_2 : Channel_42CA91F7;
	{attribute addProperty Name "WcState"}
	WcState : WcState_0B2B16F9;
	{attribute addProperty Name "InfoData"}
	InfoData : InfoData_A7436BC6;
END_STRUCT
END_TYPE

// ---- DUTs/IO/Boxes/EL2252_F49A8E92.TcDUT
{attribute 'GeneratedUsingTerminal: EL2252-0000-0017'}
{attribute addProperty BoxType "EL2252-0000-0017"}
{attribute addProperty Description "EL2252 2Ch. Dig. Output 24V, 0.5A, DC Time Stamp"}
{attribute addProperty Physics "KK"}
{attribute addProperty Id "DC_Sync_ActivateAT %Q*DC_Sync_Activate_FA2D29101DC_Sync_StartAT %Q*DC_Sync_Start_E82E92338Channel_1AT %Q*Channel_54BE63B32Channel_2AT %Q*Channel_54BE63B32ReservedEMPTY_STRUCTURE0WcStateAT %I*WcState_0B2B16F91InfoDataAT %I*InfoData_A7436BC610"}
{attribute addProperty CRC "4103769746"}
{attribute addProperty Size "24"}
TYPE EL2252_F49A8E92 EXTENDS EtcSlaveTerminalBase_947E5A46 :
STRUCT
	{attribute addProperty Name "DC_Sync_Activate"}
	DC_Sync_Activate : DC_Sync_Activate_FA2D2910;
	{attribute addProperty Name "DC_Sync_Start"}
	DC_Sync_Start : DC_Sync_Start_E82E9233;
	{attribute addProperty Name "Channel_1"}
	Channel_1 : Channel_54BE63B3;
	{attribute addProperty Name "Channel_2"}
	Channel_2 : Channel_54BE63B3;
	{attribute addProperty Name "Reserved"}
	Reserved : EMPTY_STRUCTURE;
	{attribute addProperty Name "WcState"}
	WcState : WcState_0B2B16F9;
	{attribute addProperty Name "InfoData"}
	InfoData : InfoData_A7436BC6;
END_STRUCT
END_TYPE

// ---- DUTs/IO/Boxes/EL2258_1A7A2033.TcDUT
{attribute 'GeneratedUsingTerminal: EL2258-0000-0016'}
{attribute addProperty BoxType "EL2258-0000-0016"}
{attribute addProperty Description "EL2258 8Ch. Dig Output 24V with Multi-Time-Stamp"}
{attribute addProperty Physics "KK"}
{attribute addProperty Id "MTO_Inputs_Channel_1AT %I*MTO_Inputs_Channel_53C09E8B6MTO_Inputs_Channel_2AT %I*MTO_Inputs_Channel_53C09E8B6MTO_Inputs_Channel_3AT %I*MTO_Inputs_Channel_53C09E8B6MTO_Inputs_Channel_4AT %I*MTO_Inputs_Channel_53C09E8B6MTO_Inputs_Channel_5AT %I*MTO_Inputs_Channel_53C09E8B6MTO_Inputs_Channel_6AT %I*MTO_Inputs_Channel_53C09E8B6MTO_Inputs_Channel_7AT %I*MTO_Inputs_Channel_53C09E8B6MTO_Inputs_Channel_8AT %I*MTO_Inputs_Channel_53C09E8B6MTO_Outputs_10x_Channel_1AT %Q*MTO_Outputs_10x_Channel_232E011755MTO_Outputs_10x_Channel_2AT %Q*MTO_Outputs_10x_Channel_232E011755MTO_Outputs_10x_Channel_3AT %Q*MTO_Outputs_10x_Channel_232E011755MTO_Outputs_10x_Channel_4AT %Q*MTO_Outputs_10x_Channel_232E011755MTO_Outputs_10x_Channel_5AT %Q*MTO_Outputs_10x_Channel_232E011755MTO_Outputs_10x_Channel_6AT %Q*MTO_Outputs_10x_Channel_232E011755MTO_Outputs_10x_Channel_7AT %Q*MTO_Outputs_10x_Channel_232E011755MTO_Outputs_10x_Channel_8AT %Q*MTO_Outputs_10x_Channel_232E011755WcStateAT %I*WcState_9091E0EB2InfoDataAT %I*InfoData_BEF6B88E18"}
{attribute addProperty CRC "444211251"}
{attribute addProperty Size "508"}
TYPE EL2258_1A7A2033 EXTENDS EtcSlaveTerminalBase_947E5A46 :
STRUCT
	{attribute addProperty Name "MTO_Inputs_Channel_1"}
	MTO_Inputs_Channel_1 : MTO_Inputs_Channel_53C09E8B;
	{attribute addProperty Name "MTO_Inputs_Channel_2"}
	MTO_Inputs_Channel_2 : MTO_Inputs_Channel_53C09E8B;
	{attribute addProperty Name "MTO_Inputs_Channel_3"}
	MTO_Inputs_Channel_3 : MTO_Inputs_Channel_53C09E8B;
	{attribute addProperty Name "MTO_Inputs_Channel_4"}
	MTO_Inputs_Channel_4 : MTO_Inputs_Channel_53C09E8B;
	{attribute addProperty Name "MTO_Inputs_Channel_5"}
	MTO_Inputs_Channel_5 : MTO_Inputs_Channel_53C09E8B;
	{attribute addProperty Name "MTO_Inputs_Channel_6"}
	MTO_Inputs_Channel_6 : MTO_Inputs_Channel_53C09E8B;
	{attribute addProperty Name "MTO_Inputs_Channel_7"}
	MTO_Inputs_Channel_7 : MTO_Inputs_Channel_53C09E8B;
	{attribute addProperty Name "MTO_Inputs_Channel_8"}
	MTO_Inputs_Channel_8 : MTO_Inputs_Channel_53C09E8B;
	{attribute addProperty Name "MTO_Outputs_10x_Channel_1"}
	MTO_Outputs_10x_Channel_1 : MTO_Outputs_10x_Channel_232E0117;
	{attribute addProperty Name "MTO_Outputs_10x_Channel_2"}
	MTO_Outputs_10x_Channel_2 : MTO_Outputs_10x_Channel_232E0117;
	{attribute addProperty Name "MTO_Outputs_10x_Channel_3"}
	MTO_Outputs_10x_Channel_3 : MTO_Outputs_10x_Channel_232E0117;
	{attribute addProperty Name "MTO_Outputs_10x_Channel_4"}
	MTO_Outputs_10x_Channel_4 : MTO_Outputs_10x_Channel_232E0117;
	{attribute addProperty Name "MTO_Outputs_10x_Channel_5"}
	MTO_Outputs_10x_Channel_5 : MTO_Outputs_10x_Channel_232E0117;
	{attribute addProperty Name "MTO_Outputs_10x_Channel_6"}
	MTO_Outputs_10x_Channel_6 : MTO_Outputs_10x_Channel_232E0117;
	{attribute addProperty Name "MTO_Outputs_10x_Channel_7"}
	MTO_Outputs_10x_Channel_7 : MTO_Outputs_10x_Channel_232E0117;
	{attribute addProperty Name "MTO_Outputs_10x_Channel_8"}
	MTO_Outputs_10x_Channel_8 : MTO_Outputs_10x_Channel_232E0117;
	{attribute addProperty Name "WcState"}
	WcState : WcState_9091E0EB;
	{attribute addProperty Name "InfoData"}
	InfoData : InfoData_BEF6B88E;
END_STRUCT
END_TYPE

// ---- DUTs/IO/Boxes/EL2258_41B36B91.TcDUT
{attribute 'GeneratedUsingTerminal: EL2258-0000-0017'}
{attribute addProperty BoxType "EL2258-0000-0017"}
{attribute addProperty Description "EL2258 8Ch. Dig Output 24V with Multi-Time-Stamp"}
{attribute addProperty Physics "KK"}
{attribute addProperty Id "MTO_Inputs_Channel_1AT %I*MTO_Inputs_Channel_53C09E8B6MTO_Inputs_Channel_2AT %I*MTO_Inputs_Channel_53C09E8B6MTO_Inputs_Channel_3AT %I*MTO_Inputs_Channel_53C09E8B6MTO_Inputs_Channel_4AT %I*MTO_Inputs_Channel_53C09E8B6MTO_Inputs_Channel_5AT %I*MTO_Inputs_Channel_53C09E8B6MTO_Inputs_Channel_6AT %I*MTO_Inputs_Channel_53C09E8B6MTO_Inputs_Channel_7AT %I*MTO_Inputs_Channel_53C09E8B6MTO_Inputs_Channel_8AT %I*MTO_Inputs_Channel_53C09E8B6MTO_Outputs_10x_Channel_1AT %Q*MTO_Outputs_10x_Channel_A3C0C02256MTO_Outputs_10x_Channel_2AT %Q*MTO_Outputs_10x_Channel_A3C0C02256MTO_Outputs_10x_Channel_3AT %Q*MTO_Outputs_10x_Channel_A3C0C02256MTO_Outputs_10x_Channel_4AT %Q*MTO_Outputs_10x_Channel_A3C0C02256MTO_Outputs_10x_Channel_5AT %Q*MTO_Outputs_10x_Channel_A3C0C02256MTO_Outputs_10x_Channel_6AT %Q*MTO_Outputs_10x_Channel_A3C0C02256MTO_Outputs_10x_Channel_7AT %Q*MTO_Outputs_10x_Channel_A3C0C02256MTO_Outputs_10x_Channel_8AT %Q*MTO_Outputs_10x_Channel_A3C0C02256WcStateAT %I*WcState_9091E0EB2InfoDataAT %I*InfoData_BEF6B88E18"}
{attribute addProperty CRC "1102277521"}
{attribute addProperty Size "516"}
TYPE EL2258_41B36B91 EXTENDS EtcSlaveTerminalBase_947E5A46 :
STRUCT
	{attribute addProperty Name "MTO_Inputs_Channel_1"}
	MTO_Inputs_Channel_1 : MTO_Inputs_Channel_53C09E8B;
	{attribute addProperty Name "MTO_Inputs_Channel_2"}
	MTO_Inputs_Channel_2 : MTO_Inputs_Channel_53C09E8B;
	{attribute addProperty Name "MTO_Inputs_Channel_3"}
	MTO_Inputs_Channel_3 : MTO_Inputs_Channel_53C09E8B;
	{attribute addProperty Name "MTO_Inputs_Channel_4"}
	MTO_Inputs_Channel_4 : MTO_Inputs_Channel_53C09E8B;
	{attribute addProperty Name "MTO_Inputs_Channel_5"}
	MTO_Inputs_Channel_5 : MTO_Inputs_Channel_53C09E8B;
	{attribute addProperty Name "MTO_Inputs_Channel_6"}
	MTO_Inputs_Channel_6 : MTO_Inputs_Channel_53C09E8B;
	{attribute addProperty Name "MTO_Inputs_Channel_7"}
	MTO_Inputs_Channel_7 : MTO_Inputs_Channel_53C09E8B;
	{attribute addProperty Name "MTO_Inputs_Channel_8"}
	MTO_Inputs_Channel_8 : MTO_Inputs_Channel_53C09E8B;
	{attribute addProperty Name "MTO_Outputs_10x_Channel_1"}
	MTO_Outputs_10x_Channel_1 : MTO_Outputs_10x_Channel_A3C0C022;
	{attribute addProperty Name "MTO_Outputs_10x_Channel_2"}
	MTO_Outputs_10x_Channel_2 : MTO_Outputs_10x_Channel_A3C0C022;
	{attribute addProperty Name "MTO_Outputs_10x_Channel_3"}
	MTO_Outputs_10x_Channel_3 : MTO_Outputs_10x_Channel_A3C0C022;
	{attribute addProperty Name "MTO_Outputs_10x_Channel_4"}
	MTO_Outputs_10x_Channel_4 : MTO_Outputs_10x_Channel_A3C0C022;
	{attribute addProperty Name "MTO_Outputs_10x_Channel_5"}
	MTO_Outputs_10x_Channel_5 : MTO_Outputs_10x_Channel_A3C0C022;
	{attribute addProperty Name "MTO_Outputs_10x_Channel_6"}
	MTO_Outputs_10x_Channel_6 : MTO_Outputs_10x_Channel_A3C0C022;
	{attribute addProperty Name "MTO_Outputs_10x_Channel_7"}
	MTO_Outputs_10x_Channel_7 : MTO_Outputs_10x_Channel_A3C0C022;
	{attribute addProperty Name "MTO_Outputs_10x_Channel_8"}
	MTO_Outputs_10x_Channel_8 : MTO_Outputs_10x_Channel_A3C0C022;
	{attribute addProperty Name "WcState"}
	WcState : WcState_9091E0EB;
	{attribute addProperty Name "InfoData"}
	InfoData : InfoData_BEF6B88E;
END_STRUCT
END_TYPE

// ---- DUTs/IO/Boxes/EL2262_4683CFC9.TcDUT
{attribute 'GeneratedUsingTerminal: EL2262--0000'}
{attribute addProperty BoxType "EL2262--0000"}
{attribute addProperty Description "EL2262 2Ch. Dig. Output 24V, 0.5A, DC Over Sampling"}
{attribute addProperty Physics "KK"}
{attribute addProperty Id "Cycle_CounterAT %Q*Cycle_Counter_2C2338042Sample_0AT %Q*Sample_3C4603C71WcStateAT %I*WcState_0B2B16F91InfoDataAT %I*InfoData_A7436BC610"}
{attribute addProperty CRC "1183043529"}
{attribute addProperty Size "14"}
TYPE EL2262_4683CFC9 EXTENDS EtcSlaveTerminalBase_947E5A46 :
STRUCT
	{attribute addProperty Name "Cycle_Counter"}
	Cycle_Counter : Cycle_Counter_2C233804;
	{attribute addProperty Name "Sample_0"}
	Sample_0 : Sample_3C4603C7;
	{attribute addProperty Name "WcState"}
	WcState : WcState_0B2B16F9;
	{attribute addProperty Name "InfoData"}
	InfoData : InfoData_A7436BC6;
END_STRUCT
END_TYPE

// ---- DUTs/IO/Boxes/EL2262_79C970B1.TcDUT
{attribute 'GeneratedUsingTerminal: EL2262-0000-0001'}
{attribute addProperty BoxType "EL2262-0000-0001"}
{attribute addProperty Description "EL2262 2Ch. Dig. Output 24V, 0.5A, DC Over Sampling"}
{attribute addProperty Physics "KK"}
{attribute addProperty Id "CycCount0AT %Q*CycCount0_2C2338042Sample0_0AT %Q*Sample_0023574C1GapAT %I*EMPTY_STRUCTURE0CycCount1AT %Q*CycCount1_2C2338042Sample1_0AT %Q*Sample_07D5B44A1Gap_1AT %I*EMPTY_STRUCTURE0WcStateAT %I*WcState_0B2B16F91InfoDataAT %I*InfoData_A7436BC610"}
{attribute addProperty CRC "2043244721"}
{attribute addProperty Size "17"}
TYPE EL2262_79C970B1 EXTENDS EtcSlaveTerminalBase_947E5A46 :
STRUCT
	{attribute addProperty Name "CycCount0"}
	CycCount0 : CycCount0_2C233804;
	{attribute addProperty Name "Sample0_0"}
	Sample0_0 : Sample_0023574C;
	{attribute addProperty Name "Gap"}
	Gap : EMPTY_STRUCTURE;
	{attribute addProperty Name "CycCount1"}
	CycCount1 : CycCount1_2C233804;
	{attribute addProperty Name "Sample1_0"}
	Sample1_0 : Sample_07D5B44A;
	{attribute addProperty Name "Gap_1"}
	Gap_1 : EMPTY_STRUCTURE;
	{attribute addProperty Name "WcState"}
	WcState : WcState_0B2B16F9;
	{attribute addProperty Name "InfoData"}
	InfoData : InfoData_A7436BC6;
END_STRUCT
END_TYPE

// ---- DUTs/IO/Boxes/EL2262_147DB6E1.TcDUT
{attribute 'GeneratedUsingTerminal: EL2262-0000-0002'}
{attribute addProperty BoxType "EL2262-0000-0002"}
{attribute addProperty Description "EL2262 2Ch. Dig. Output 24V, 1µs, DC Oversample"}
{attribute addProperty Physics "KK"}
{attribute addProperty Id "CycCount0AT %Q*CycCount0_AF431CE02Sample0_0AT %Q*Sample_0023574C1Sample0_1AT %Q*Sample_0023574C1Sample0_2AT %Q*Sample_0023574C1Sample0_3AT %Q*Sample_0023574C1Sample0_4AT %Q*Sample_0023574C1Sample0_5AT %Q*Sample_0023574C1Sample0_6AT %Q*Sample_0023574C1Sample0_7AT %Q*Sample_0023574C1Sample0_8AT %Q*Sample_0023574C1Sample0_9AT %Q*Sample_0023574C1GapAT %I*EMPTY_STRUCTURE0CycCount1AT %Q*CycCount1_A8B5FFE62Sample1_0AT %Q*Sample_07D5B44A1Sample1_1AT %Q*Sample_07D5B44A1Sample1_2AT %Q*Sample_07D5B44A1Sample1_3AT %Q*Sample_07D5B44A1Sample1_4AT %Q*Sample_07D5B44A1Sample1_5AT %Q*Sample_07D5B44A1Sample1_6AT %Q*Sample_07D5B44A1Sample1_7AT %Q*Sample_07D5B44A1Sample1_8AT %Q*Sample_07D5B44A1Sample1_9AT %Q*Sample_07D5B44A1Gap_1AT %I*EMPTY_STRUCTURE0WcStateAT %I*WcState_0B2B16F91InfoDataAT %I*InfoData_A7436BC610"}
{attribute addProperty CRC "343783137"}
{attribute addProperty Size "35"}
TYPE EL2262_147DB6E1 EXTENDS EtcSlaveTerminalBase_947E5A46 :
STRUCT
	{attribute addProperty Name "CycCount0"}
	CycCount0 : CycCount0_AF431CE0;
	{attribute addProperty Name "Sample0_0"}
	Sample0_0 : Sample_0023574C;
	{attribute addProperty Name "Sample0_1"}
	Sample0_1 : Sample_0023574C;
	{attribute addProperty Name "Sample0_2"}
	Sample0_2 : Sample_0023574C;
	{attribute addProperty Name "Sample0_3"}
	Sample0_3 : Sample_0023574C;
	{attribute addProperty Name "Sample0_4"}
	Sample0_4 : Sample_0023574C;
	{attribute addProperty Name "Sample0_5"}
	Sample0_5 : Sample_0023574C;
	{attribute addProperty Name "Sample0_6"}
	Sample0_6 : Sample_0023574C;
	{attribute addProperty Name "Sample0_7"}
	Sample0_7 : Sample_0023574C;
	{attribute addProperty Name "Sample0_8"}
	Sample0_8 : Sample_0023574C;
	{attribute addProperty Name "Sample0_9"}
	Sample0_9 : Sample_0023574C;
	{attribute addProperty Name "Gap"}
	Gap : EMPTY_STRUCTURE;
	{attribute addProperty Name "CycCount1"}
	CycCount1 : CycCount1_A8B5FFE6;
	{attribute addProperty Name "Sample1_0"}
	Sample1_0 : Sample_07D5B44A;
	{attribute addProperty Name "Sample1_1"}
	Sample1_1 : Sample_07D5B44A;
	{attribute addProperty Name "Sample1_2"}
	Sample1_2 : Sample_07D5B44A;
	{attribute addProperty Name "Sample1_3"}
	Sample1_3 : Sample_07D5B44A;
	{attribute addProperty Name "Sample1_4"}
	Sample1_4 : Sample_07D5B44A;
	{attribute addProperty Name "Sample1_5"}
	Sample1_5 : Sample_07D5B44A;
	{attribute addProperty Name "Sample1_6"}
	Sample1_6 : Sample_07D5B44A;
	{attribute addProperty Name "Sample1_7"}
	Sample1_7 : Sample_07D5B44A;
	{attribute addProperty Name "Sample1_8"}
	Sample1_8 : Sample_07D5B44A;
	{attribute addProperty Name "Sample1_9"}
	Sample1_9 : Sample_07D5B44A;
	{attribute addProperty Name "Gap_1"}
	Gap_1 : EMPTY_STRUCTURE;
	{attribute addProperty Name "WcState"}
	WcState : WcState_0B2B16F9;
	{attribute addProperty Name "InfoData"}
	InfoData : InfoData_A7436BC6;
END_STRUCT
END_TYPE

// ---- DUTs/IO/Boxes/EL2262_9619875D.TcDUT
{attribute 'GeneratedUsingTerminal: EL2262-0000-0004'}
{attribute addProperty BoxType "EL2262-0000-0004"}
{attribute addProperty Description "EL2262 2Ch. Dig. Output 24V, 1µs, DC Oversample"}
{attribute addProperty Physics "KK"}
{attribute addProperty Id "StartTimeNextOutputAT %I*StartTimeNextOutput_228767F44CycCount0AT %Q*CycCount0_AF431CE02Sample0_0AT %Q*Sample_0023574C1Sample0_1AT %Q*Sample_0023574C1Sample0_2AT %Q*Sample_0023574C1Sample0_3AT %Q*Sample_0023574C1Sample0_4AT %Q*Sample_0023574C1Sample0_5AT %Q*Sample_0023574C1Sample0_6AT %Q*Sample_0023574C1Sample0_7AT %Q*Sample_0023574C1Sample0_8AT %Q*Sample_0023574C1Sample0_9AT %Q*Sample_0023574C1GapAT %I*EMPTY_STRUCTURE0CycCount1AT %Q*CycCount1_A8B5FFE62Sample1_0AT %Q*Sample_07D5B44A1Sample1_1AT %Q*Sample_07D5B44A1Sample1_2AT %Q*Sample_07D5B44A1Sample1_3AT %Q*Sample_07D5B44A1Sample1_4AT %Q*Sample_07D5B44A1Sample1_5AT %Q*Sample_07D5B44A1Sample1_6AT %Q*Sample_07D5B44A1Sample1_7AT %Q*Sample_07D5B44A1Sample1_8AT %Q*Sample_07D5B44A1Sample1_9AT %Q*Sample_07D5B44A1Gap_1AT %I*EMPTY_STRUCTURE0WcStateAT %I*WcState_9091E0EB2InfoDataAT %I*InfoData_A7436BC610"}
{attribute addProperty CRC "2518255453"}
{attribute addProperty Size "40"}
TYPE EL2262_9619875D EXTENDS EtcSlaveTerminalBase_947E5A46 :
STRUCT
	{attribute addProperty Name "StartTimeNextOutput"}
	StartTimeNextOutput : StartTimeNextOutput_228767F4;
	{attribute addProperty Name "CycCount0"}
	CycCount0 : CycCount0_AF431CE0;
	{attribute addProperty Name "Sample0_0"}
	Sample0_0 : Sample_0023574C;
	{attribute addProperty Name "Sample0_1"}
	Sample0_1 : Sample_0023574C;
	{attribute addProperty Name "Sample0_2"}
	Sample0_2 : Sample_0023574C;
	{attribute addProperty Name "Sample0_3"}
	Sample0_3 : Sample_0023574C;
	{attribute addProperty Name "Sample0_4"}
	Sample0_4 : Sample_0023574C;
	{attribute addProperty Name "Sample0_5"}
	Sample0_5 : Sample_0023574C;
	{attribute addProperty Name "Sample0_6"}
	Sample0_6 : Sample_0023574C;
	{attribute addProperty Name "Sample0_7"}
	Sample0_7 : Sample_0023574C;
	{attribute addProperty Name "Sample0_8"}
	Sample0_8 : Sample_0023574C;
	{attribute addProperty Name "Sample0_9"}
	Sample0_9 : Sample_0023574C;
	{attribute addProperty Name "Gap"}
	Gap : EMPTY_STRUCTURE;
	{attribute addProperty Name "CycCount1"}
	CycCount1 : CycCount1_A8B5FFE6;
	{attribute addProperty Name "Sample1_0"}
	Sample1_0 : Sample_07D5B44A;
	{attribute addProperty Name "Sample1_1"}
	Sample1_1 : Sample_07D5B44A;
	{attribute addProperty Name "Sample1_2"}
	Sample1_2 : Sample_07D5B44A;
	{attribute addProperty Name "Sample1_3"}
	Sample1_3 : Sample_07D5B44A;
	{attribute addProperty Name "Sample1_4"}
	Sample1_4 : Sample_07D5B44A;
	{attribute addProperty Name "Sample1_5"}
	Sample1_5 : Sample_07D5B44A;
	{attribute addProperty Name "Sample1_6"}
	Sample1_6 : Sample_07D5B44A;
	{attribute addProperty Name "Sample1_7"}
	Sample1_7 : Sample_07D5B44A;
	{attribute addProperty Name "Sample1_8"}
	Sample1_8 : Sample_07D5B44A;
	{attribute addProperty Name "Sample1_9"}
	Sample1_9 : Sample_07D5B44A;
	{attribute addProperty Name "Gap_1"}
	Gap_1 : EMPTY_STRUCTURE;
	{attribute addProperty Name "WcState"}
	WcState : WcState_9091E0EB;
	{attribute addProperty Name "InfoData"}
	InfoData : InfoData_A7436BC6;
END_STRUCT
END_TYPE

// ---- DUTs/IO/Boxes/EL2602_B0214940.TcDUT
{attribute 'GeneratedUsingTerminal: EL2602-0000-0016'}
{attribute addProperty BoxType "EL2602-0000-0016"}
{attribute addProperty Description "EL2602 2Ch. Relay Output, NO (230V AC / 30V DC)"}
{attribute addProperty Physics "KK"}
{attribute addProperty Id "Channel_1AT %Q*Channel_42CA91F71Channel_2AT %Q*Channel_42CA91F71WcStateAT %I*WcState_0B2B16F91InfoDataAT %I*InfoData_6F19DB2B2"}
{attribute addProperty CRC "2954971456"}
{attribute addProperty Size "5"}
TYPE EL2602_B0214940 EXTENDS EtcSlaveTerminalBase_947E5A46 :
STRUCT
	{attribute addProperty Name "Channel_1"}
	Channel_1 : Channel_42CA91F7;
	{attribute addProperty Name "Channel_2"}
	Channel_2 : Channel_42CA91F7;
	{attribute addProperty Name "WcState"}
	WcState : WcState_0B2B16F9;
	{attribute addProperty Name "InfoData"}
	InfoData : InfoData_6F19DB2B;
END_STRUCT
END_TYPE

// ---- DUTs/IO/Boxes/EL2602_47E63F27.TcDUT
{attribute 'GeneratedUsingTerminal: EL2602-0010-0016'}
{attribute addProperty BoxType "EL2602-0010-0016"}
{attribute addProperty Description "EL2602-0010 2Ch. Relay Output + ZCD, NO (230V AC / 30V DC)"}
{attribute addProperty Physics "KK"}
{attribute addProperty Id "InputsAT %I*Inputs_298FB92D1Channel_1AT %Q*Channel_42CA91F71Channel_2AT %Q*Channel_42CA91F71WcStateAT %I*WcState_9091E0EB2InfoDataAT %I*InfoData_6F19DB2B2"}
{attribute addProperty CRC "1206271783"}
{attribute addProperty Size "7"}
TYPE EL2602_47E63F27 EXTENDS EtcSlaveTerminalBase_947E5A46 :
STRUCT
	{attribute addProperty Name "Inputs"}
	Inputs : Inputs_298FB92D;
	{attribute addProperty Name "Channel_1"}
	Channel_1 : Channel_42CA91F7;
	{attribute addProperty Name "Channel_2"}
	Channel_2 : Channel_42CA91F7;
	{attribute addProperty Name "WcState"}
	WcState : WcState_9091E0EB;
	{attribute addProperty Name "InfoData"}
	InfoData : InfoData_6F19DB2B;
END_STRUCT
END_TYPE

// ---- DUTs/IO/Boxes/EL2612_B0214940.TcDUT
{attribute 'GeneratedUsingTerminal: EL2612-0000-0016'}
{attribute addProperty BoxType "EL2612-0000-0016"}
{attribute addProperty Description "EL2612 2Ch. Relay Output, CO (125V AC / 30V DC)"}
{attribute addProperty Physics "KK"}
{attribute addProperty Id "Channel_1AT %Q*Channel_42CA91F71Channel_2AT %Q*Channel_42CA91F71WcStateAT %I*WcState_0B2B16F91InfoDataAT %I*InfoData_6F19DB2B2"}
{attribute addProperty CRC "2954971456"}
{attribute addProperty Size "5"}
TYPE EL2612_B0214940 EXTENDS EtcSlaveTerminalBase_947E5A46 :
STRUCT
	{attribute addProperty Name "Channel_1"}
	Channel_1 : Channel_42CA91F7;
	{attribute addProperty Name "Channel_2"}
	Channel_2 : Channel_42CA91F7;
	{attribute addProperty Name "WcState"}
	WcState : WcState_0B2B16F9;
	{attribute addProperty Name "InfoData"}
	InfoData : InfoData_6F19DB2B;
END_STRUCT
END_TYPE

// ---- DUTs/IO/Boxes/EL2622_B0214940.TcDUT
{attribute 'GeneratedUsingTerminal: EL2622-0000-0016'}
{attribute addProperty BoxType "EL2622-0000-0016"}
{attribute addProperty Description "EL2622 2Ch. Relay Output, NO (230V AC / 30V DC)"}
{attribute addProperty Physics "KK"}
{attribute addProperty Id "Channel_1AT %Q*Channel_42CA91F71Channel_2AT %Q*Channel_42CA91F71WcStateAT %I*WcState_0B2B16F91InfoDataAT %I*InfoData_6F19DB2B2"}
{attribute addProperty CRC "2954971456"}
{attribute addProperty Size "5"}
TYPE EL2622_B0214940 EXTENDS EtcSlaveTerminalBase_947E5A46 :
STRUCT
	{attribute addProperty Name "Channel_1"}
	Channel_1 : Channel_42CA91F7;
	{attribute addProperty Name "Channel_2"}
	Channel_2 : Channel_42CA91F7;
	{attribute addProperty Name "WcState"}
	WcState : WcState_0B2B16F9;
	{attribute addProperty Name "InfoData"}
	InfoData : InfoData_6F19DB2B;
END_STRUCT
END_TYPE

// ---- DUTs/IO/Boxes/EL2622_47E63F27.TcDUT
{attribute 'GeneratedUsingTerminal: EL2622-0010-0016'}
{attribute addProperty BoxType "EL2622-0010-0016"}
{attribute addProperty Description "EL2622-0010 2Ch. Relay Output + ZCD, NO (230V AC / 30V DC)"}
{attribute addProperty Physics "KK"}
{attribute addProperty Id "InputsAT %I*Inputs_298FB92D1Channel_1AT %Q*Channel_42CA91F71Channel_2AT %Q*Channel_42CA91F71WcStateAT %I*WcState_9091E0EB2InfoDataAT %I*InfoData_6F19DB2B2"}
{attribute addProperty CRC "1206271783"}
{attribute addProperty Size "7"}
TYPE EL2622_47E63F27 EXTENDS EtcSlaveTerminalBase_947E5A46 :
STRUCT
	{attribute addProperty Name "Inputs"}
	Inputs : Inputs_298FB92D;
	{attribute addProperty Name "Channel_1"}
	Channel_1 : Channel_42CA91F7;
	{attribute addProperty Name "Channel_2"}
	Channel_2 : Channel_42CA91F7;
	{attribute addProperty Name "WcState"}
	WcState : WcState_9091E0EB;
	{attribute addProperty Name "InfoData"}
	InfoData : InfoData_6F19DB2B;
END_STRUCT
END_TYPE

// ---- DUTs/IO/Boxes/EL2624_7B64371E.TcDUT
{attribute 'GeneratedUsingTerminal: EL2624-0000-0016'}
{attribute addProperty BoxType "EL2624-0000-0016"}
{attribute addProperty Description "EL2624 4Ch. Relay Output, NO (125V AC / 30V DC)"}
{attribute addProperty Physics "KK"}
{attribute addProperty Id "Channel_1AT %Q*Channel_42CA91F71Channel_2AT %Q*Channel_42CA91F71Channel_3AT %Q*Channel_42CA91F71Channel_4AT %Q*Channel_42CA91F71WcStateAT %I*WcState_0B2B16F91InfoDataAT %I*InfoData_6F19DB2B2"}
{attribute addProperty CRC "2070165278"}
{attribute addProperty Size "7"}
TYPE EL2624_7B64371E EXTENDS EtcSlaveTerminalBase_947E5A46 :
STRUCT
	{attribute addProperty Name "Channel_1"}
	Channel_1 : Channel_42CA91F7;
	{attribute addProperty Name "Channel_2"}
	Channel_2 : Channel_42CA91F7;
	{attribute addProperty Name "Channel_3"}
	Channel_3 : Channel_42CA91F7;
	{attribute addProperty Name "Channel_4"}
	Channel_4 : Channel_42CA91F7;
	{attribute addProperty Name "WcState"}
	WcState : WcState_0B2B16F9;
	{attribute addProperty Name "InfoData"}
	InfoData : InfoData_6F19DB2B;
END_STRUCT
END_TYPE

// ---- DUTs/IO/Boxes/EL2634_7B64371E.TcDUT
{attribute 'GeneratedUsingTerminal: EL2634-0000-0016'}
{attribute addProperty BoxType "EL2634-0000-0016"}
{attribute addProperty Description "EL2634 4Ch. Relay Output, NO (250V AC / 30V DC)"}
{attribute addProperty Physics "KK"}
{attribute addProperty Id "Channel_1AT %Q*Channel_42CA91F71Channel_2AT %Q*Channel_42CA91F71Channel_3AT %Q*Channel_42CA91F71Channel_4AT %Q*Channel_42CA91F71WcStateAT %I*WcState_0B2B16F91InfoDataAT %I*InfoData_6F19DB2B2"}
{attribute addProperty CRC "2070165278"}
{attribute addProperty Size "7"}
TYPE EL2634_7B64371E EXTENDS EtcSlaveTerminalBase_947E5A46 :
STRUCT
	{attribute addProperty Name "Channel_1"}
	Channel_1 : Channel_42CA91F7;
	{attribute addProperty Name "Channel_2"}
	Channel_2 : Channel_42CA91F7;
	{attribute addProperty Name "Channel_3"}
	Channel_3 : Channel_42CA91F7;
	{attribute addProperty Name "Channel_4"}
	Channel_4 : Channel_42CA91F7;
	{attribute addProperty Name "WcState"}
	WcState : WcState_0B2B16F9;
	{attribute addProperty Name "InfoData"}
	InfoData : InfoData_6F19DB2B;
END_STRUCT
END_TYPE

// ---- DUTs/IO/Boxes/EL2642_C5F9ACE7.TcDUT
{attribute 'GeneratedUsingTerminal: EL2642-0000-0016'}
{attribute addProperty BoxType "EL2642-0000-0016"}
{attribute addProperty Description "EL2642 2Ch. Multiplexer Ausgang 1x4 Reed-Relais 48V AC/DC, 1A, potential-free"}
{attribute addProperty Physics "KK"}
{attribute addProperty Id "DO_Inputs_DeviceAT %I*DO_Inputs_Device_4A9049C53DO_Group_1_OutputsAT %Q*DO_Group_1_Outputs_59D8C01C4DO_Group_2_OutputsAT %Q*DO_Group_2_Outputs_828082884WcStateAT %I*WcState_9091E0EB2InfoDataAT %I*InfoData_BEF6B88E18"}
{attribute addProperty CRC "3321474279"}
{attribute addProperty Size "31"}
TYPE EL2642_C5F9ACE7 EXTENDS EtcSlaveTerminalBase_947E5A46 :
STRUCT
	{attribute addProperty Name "DO_Inputs_Device"}
	DO_Inputs_Device : DO_Inputs_Device_4A9049C5;
	{attribute addProperty Name "DO_Group_1_Outputs"}
	DO_Group_1_Outputs : DO_Group_1_Outputs_59D8C01C;
	{attribute addProperty Name "DO_Group_2_Outputs"}
	DO_Group_2_Outputs : DO_Group_2_Outputs_82808288;
	{attribute addProperty Name "WcState"}
	WcState : WcState_9091E0EB;
	{attribute addProperty Name "InfoData"}
	InfoData : InfoData_BEF6B88E;
END_STRUCT
END_TYPE

// ---- DUTs/IO/Boxes/EL2652_B0214940.TcDUT
{attribute 'GeneratedUsingTerminal: EL2652-0000-0016'}
{attribute addProperty BoxType "EL2652-0000-0016"}
{attribute addProperty Description "EL2652 2Ch. Relay Output, CO (230V AC / 30V DC)"}
{attribute addProperty Physics "KK"}
{attribute addProperty Id "Channel_1AT %Q*Channel_42CA91F71Channel_2AT %Q*Channel_42CA91F71WcStateAT %I*WcState_0B2B16F91InfoDataAT %I*InfoData_6F19DB2B2"}
{attribute addProperty CRC "2954971456"}
{attribute addProperty Size "5"}
TYPE EL2652_B0214940 EXTENDS EtcSlaveTerminalBase_947E5A46 :
STRUCT
	{attribute addProperty Name "Channel_1"}
	Channel_1 : Channel_42CA91F7;
	{attribute addProperty Name "Channel_2"}
	Channel_2 : Channel_42CA91F7;
	{attribute addProperty Name "WcState"}
	WcState : WcState_0B2B16F9;
	{attribute addProperty Name "InfoData"}
	InfoData : InfoData_6F19DB2B;
END_STRUCT
END_TYPE

// ---- DUTs/IO/Boxes/EL2712_B0214940.TcDUT
{attribute 'GeneratedUsingTerminal: EL2712-0000-0016'}
{attribute addProperty BoxType "EL2712-0000-0016"}
{attribute addProperty Description "EL2712 2Ch. Triac Output 12..230V AC, 0.5A"}
{attribute addProperty Physics "KK"}
{attribute addProperty Id "Channel_1AT %Q*Channel_42CA91F71Channel_2AT %Q*Channel_42CA91F71WcStateAT %I*WcState_0B2B16F91InfoDataAT %I*InfoData_6F19DB2B2"}
{attribute addProperty CRC "2954971456"}
{attribute addProperty Size "5"}
TYPE EL2712_B0214940 EXTENDS EtcSlaveTerminalBase_947E5A46 :
STRUCT
	{attribute addProperty Name "Channel_1"}
	Channel_1 : Channel_42CA91F7;
	{attribute addProperty Name "Channel_2"}
	Channel_2 : Channel_42CA91F7;
	{attribute addProperty Name "WcState"}
	WcState : WcState_0B2B16F9;
	{attribute addProperty Name "InfoData"}
	InfoData : InfoData_6F19DB2B;
END_STRUCT
END_TYPE

// ---- DUTs/IO/Boxes/EL2722_B0214940.TcDUT
{attribute 'GeneratedUsingTerminal: EL2722-0000-0016'}
{attribute addProperty BoxType "EL2722-0000-0016"}
{attribute addProperty Description "EL2722 2Ch. Triac Output 12..230V AC, 1.0A, mutually locked"}
{attribute addProperty Physics "KK"}
{attribute addProperty Id "Channel_1AT %Q*Channel_42CA91F71Channel_2AT %Q*Channel_42CA91F71WcStateAT %I*WcState_0B2B16F91InfoDataAT %I*InfoData_6F19DB2B2"}
{attribute addProperty CRC "2954971456"}
{attribute addProperty Size "5"}
TYPE EL2722_B0214940 EXTENDS EtcSlaveTerminalBase_947E5A46 :
STRUCT
	{attribute addProperty Name "Channel_1"}
	Channel_1 : Channel_42CA91F7;
	{attribute addProperty Name "Channel_2"}
	Channel_2 : Channel_42CA91F7;
	{attribute addProperty Name "WcState"}
	WcState : WcState_0B2B16F9;
	{attribute addProperty Name "InfoData"}
	InfoData : InfoData_6F19DB2B;
END_STRUCT
END_TYPE

// ---- DUTs/IO/Boxes/EL2732_B0214940.TcDUT
{attribute 'GeneratedUsingTerminal: EL2732-0000-0016'}
{attribute addProperty BoxType "EL2732-0000-0016"}
{attribute addProperty Description "EL2732 2Ch. Triac Output 12..230V AC, 0.5A, no power contacts"}
{attribute addProperty Physics "KK"}
{attribute addProperty Id "Channel_1AT %Q*Channel_42CA91F71Channel_2AT %Q*Channel_42CA91F71WcStateAT %I*WcState_0B2B16F91InfoDataAT %I*InfoData_6F19DB2B2"}
{attribute addProperty CRC "2954971456"}
{attribute addProperty Size "5"}
TYPE EL2732_B0214940 EXTENDS EtcSlaveTerminalBase_947E5A46 :
STRUCT
	{attribute addProperty Name "Channel_1"}
	Channel_1 : Channel_42CA91F7;
	{attribute addProperty Name "Channel_2"}
	Channel_2 : Channel_42CA91F7;
	{attribute addProperty Name "WcState"}
	WcState : WcState_0B2B16F9;
	{attribute addProperty Name "InfoData"}
	InfoData : InfoData_6F19DB2B;
END_STRUCT
END_TYPE

// ---- DUTs/IO/Boxes/EL2784_7B64371E.TcDUT
{attribute 'GeneratedUsingTerminal: EL2784-0000-0016'}
{attribute addProperty BoxType "EL2784-0000-0016"}
{attribute addProperty Description "EL2784 4Ch. Dig. Output 24V AC/DC, 2A, short-circuit-proof"}
{attribute addProperty Physics "KK"}
{attribute addProperty Id "Channel_1AT %Q*Channel_42CA91F71Channel_2AT %Q*Channel_42CA91F71Channel_3AT %Q*Channel_42CA91F71Channel_4AT %Q*Channel_42CA91F71WcStateAT %I*WcState_0B2B16F91InfoDataAT %I*InfoData_6F19DB2B2"}
{attribute addProperty CRC "2070165278"}
{attribute addProperty Size "7"}
TYPE EL2784_7B64371E EXTENDS EtcSlaveTerminalBase_947E5A46 :
STRUCT
	{attribute addProperty Name "Channel_1"}
	Channel_1 : Channel_42CA91F7;
	{attribute addProperty Name "Channel_2"}
	Channel_2 : Channel_42CA91F7;
	{attribute addProperty Name "Channel_3"}
	Channel_3 : Channel_42CA91F7;
	{attribute addProperty Name "Channel_4"}
	Channel_4 : Channel_42CA91F7;
	{attribute addProperty Name "WcState"}
	WcState : WcState_0B2B16F9;
	{attribute addProperty Name "InfoData"}
	InfoData : InfoData_6F19DB2B;
END_STRUCT
END_TYPE

// ---- DUTs/IO/Boxes/EL2788_E2806B95.TcDUT
{attribute 'GeneratedUsingTerminal: EL2788-0000-0016'}
{attribute addProperty BoxType "EL2788-0000-0016"}
{attribute addProperty Description "EL2788 8Ch. Dig. Output 24V AC/DC, 2A"}
{attribute addProperty Physics "KK"}
{attribute addProperty Id "Channel_1AT %Q*Channel_42CA91F71Channel_2AT %Q*Channel_42CA91F71Channel_3AT %Q*Channel_42CA91F71Channel_4AT %Q*Channel_42CA91F71Channel_5AT %Q*Channel_42CA91F71Channel_6AT %Q*Channel_42CA91F71Channel_7AT %Q*Channel_42CA91F71Channel_8AT %Q*Channel_42CA91F71WcStateAT %I*WcState_0B2B16F91InfoDataAT %I*InfoData_6F19DB2B2"}
{attribute addProperty CRC "3800066965"}
{attribute addProperty Size "11"}
TYPE EL2788_E2806B95 EXTENDS EtcSlaveTerminalBase_947E5A46 :
STRUCT
	{attribute addProperty Name "Channel_1"}
	Channel_1 : Channel_42CA91F7;
	{attribute addProperty Name "Channel_2"}
	Channel_2 : Channel_42CA91F7;
	{attribute addProperty Name "Channel_3"}
	Channel_3 : Channel_42CA91F7;
	{attribute addProperty Name "Channel_4"}
	Channel_4 : Channel_42CA91F7;
	{attribute addProperty Name "Channel_5"}
	Channel_5 : Channel_42CA91F7;
	{attribute addProperty Name "Channel_6"}
	Channel_6 : Channel_42CA91F7;
	{attribute addProperty Name "Channel_7"}
	Channel_7 : Channel_42CA91F7;
	{attribute addProperty Name "Channel_8"}
	Channel_8 : Channel_42CA91F7;
	{attribute addProperty Name "WcState"}
	WcState : WcState_0B2B16F9;
	{attribute addProperty Name "InfoData"}
	InfoData : InfoData_6F19DB2B;
END_STRUCT
END_TYPE

// ---- DUTs/IO/Boxes/EL2794_7B64371E.TcDUT
{attribute 'GeneratedUsingTerminal: EL2794-0000-0016'}
{attribute addProperty BoxType "EL2794-0000-0016"}
{attribute addProperty Description "EL2794 4Ch. Dig. Output 24V AC/DC, 2A, short-circuit-proof"}
{attribute addProperty Physics "KK"}
{attribute addProperty Id "Channel_1AT %Q*Channel_42CA91F71Channel_2AT %Q*Channel_42CA91F71Channel_3AT %Q*Channel_42CA91F71Channel_4AT %Q*Channel_42CA91F71WcStateAT %I*WcState_0B2B16F91InfoDataAT %I*InfoData_6F19DB2B2"}
{attribute addProperty CRC "2070165278"}
{attribute addProperty Size "7"}
TYPE EL2794_7B64371E EXTENDS EtcSlaveTerminalBase_947E5A46 :
STRUCT
	{attribute addProperty Name "Channel_1"}
	Channel_1 : Channel_42CA91F7;
	{attribute addProperty Name "Channel_2"}
	Channel_2 : Channel_42CA91F7;
	{attribute addProperty Name "Channel_3"}
	Channel_3 : Channel_42CA91F7;
	{attribute addProperty Name "Channel_4"}
	Channel_4 : Channel_42CA91F7;
	{attribute addProperty Name "WcState"}
	WcState : WcState_0B2B16F9;
	{attribute addProperty Name "InfoData"}
	InfoData : InfoData_6F19DB2B;
END_STRUCT
END_TYPE

// ---- DUTs/IO/Boxes/EL2798_E2806B95.TcDUT
{attribute 'GeneratedUsingTerminal: EL2798-0000-0016'}
{attribute addProperty BoxType "EL2798-0000-0016"}
{attribute addProperty Description "EL2798 8Ch. Dig. Output 24V AC/DC, 2A, potential-free"}
{attribute addProperty Physics "KK"}
{attribute addProperty Id "Channel_1AT %Q*Channel_42CA91F71Channel_2AT %Q*Channel_42CA91F71Channel_3AT %Q*Channel_42CA91F71Channel_4AT %Q*Channel_42CA91F71Channel_5AT %Q*Channel_42CA91F71Channel_6AT %Q*Channel_42CA91F71Channel_7AT %Q*Channel_42CA91F71Channel_8AT %Q*Channel_42CA91F71WcStateAT %I*WcState_0B2B16F91InfoDataAT %I*InfoData_6F19DB2B2"}
{attribute addProperty CRC "3800066965"}
{attribute addProperty Size "11"}
TYPE EL2798_E2806B95 EXTENDS EtcSlaveTerminalBase_947E5A46 :
STRUCT
	{attribute addProperty Name "Channel_1"}
	Channel_1 : Channel_42CA91F7;
	{attribute addProperty Name "Channel_2"}
	Channel_2 : Channel_42CA91F7;
	{attribute addProperty Name "Channel_3"}
	Channel_3 : Channel_42CA91F7;
	{attribute addProperty Name "Channel_4"}
	Channel_4 : Channel_42CA91F7;
	{attribute addProperty Name "Channel_5"}
	Channel_5 : Channel_42CA91F7;
	{attribute addProperty Name "Channel_6"}
	Channel_6 : Channel_42CA91F7;
	{attribute addProperty Name "Channel_7"}
	Channel_7 : Channel_42CA91F7;
	{attribute addProperty Name "Channel_8"}
	Channel_8 : Channel_42CA91F7;
	{attribute addProperty Name "WcState"}
	WcState : WcState_0B2B16F9;
	{attribute addProperty Name "InfoData"}
	InfoData : InfoData_6F19DB2B;
END_STRUCT
END_TYPE

// ---- DUTs/IO/Boxes/EL2808_E2806B95.TcDUT
{attribute 'GeneratedUsingTerminal: EL2808-0000-0016'}
{attribute addProperty BoxType "EL2808-0000-0016"}
{attribute addProperty Description "EL2808 8Ch. Dig. Output 24V, 0.5A"}
{attribute addProperty Physics "KK"}
{attribute addProperty Id "Channel_1AT %Q*Channel_42CA91F71Channel_2AT %Q*Channel_42CA91F71Channel_3AT %Q*Channel_42CA91F71Channel_4AT %Q*Channel_42CA91F71Channel_5AT %Q*Channel_42CA91F71Channel_6AT %Q*Channel_42CA91F71Channel_7AT %Q*Channel_42CA91F71Channel_8AT %Q*Channel_42CA91F71WcStateAT %I*WcState_0B2B16F91InfoDataAT %I*InfoData_6F19DB2B2"}
{attribute addProperty CRC "3800066965"}
{attribute addProperty Size "11"}
TYPE EL2808_E2806B95 EXTENDS EtcSlaveTerminalBase_947E5A46 :
STRUCT
	{attribute addProperty Name "Channel_1"}
	Channel_1 : Channel_42CA91F7;
	{attribute addProperty Name "Channel_2"}
	Channel_2 : Channel_42CA91F7;
	{attribute addProperty Name "Channel_3"}
	Channel_3 : Channel_42CA91F7;
	{attribute addProperty Name "Channel_4"}
	Channel_4 : Channel_42CA91F7;
	{attribute addProperty Name "Channel_5"}
	Channel_5 : Channel_42CA91F7;
	{attribute addProperty Name "Channel_6"}
	Channel_6 : Channel_42CA91F7;
	{attribute addProperty Name "Channel_7"}
	Channel_7 : Channel_42CA91F7;
	{attribute addProperty Name "Channel_8"}
	Channel_8 : Channel_42CA91F7;
	{attribute addProperty Name "WcState"}
	WcState : WcState_0B2B16F9;
	{attribute addProperty Name "InfoData"}
	InfoData : InfoData_6F19DB2B;
END_STRUCT
END_TYPE

// ---- DUTs/IO/Boxes/EL2809_2B6483BD.TcDUT
{attribute 'GeneratedUsingTerminal: EL2809-0000-0016'}
{attribute addProperty BoxType "EL2809-0000-0016"}
{attribute addProperty Description "EL2809 16Ch. Dig. Output 24V, 0.5A"}
{attribute addProperty Physics "KK"}
{attribute addProperty Id "Channel_1AT %Q*Channel_42CA91F71Channel_2AT %Q*Channel_42CA91F71Channel_3AT %Q*Channel_42CA91F71Channel_4AT %Q*Channel_42CA91F71Channel_5AT %Q*Channel_42CA91F71Channel_6AT %Q*Channel_42CA91F71Channel_7AT %Q*Channel_42CA91F71Channel_8AT %Q*Channel_42CA91F71Channel_9AT %Q*Channel_42CA91F71Channel_10AT %Q*Channel_42CA91F71Channel_11AT %Q*Channel_42CA91F71Channel_12AT %Q*Channel_42CA91F71Channel_13AT %Q*Channel_42CA91F71Channel_14AT %Q*Channel_42CA91F71Channel_15AT %Q*Channel_42CA91F71Channel_16AT %Q*Channel_42CA91F71WcStateAT %I*WcState_0B2B16F91InfoDataAT %I*InfoData_6F19DB2B2"}
{attribute addProperty CRC "728007613"}
{attribute addProperty Size "19"}
TYPE EL2809_2B6483BD EXTENDS EtcSlaveTerminalBase_947E5A46 :
STRUCT
	{attribute addProperty Name "Channel_1"}
	Channel_1 : Channel_42CA91F7;
	{attribute addProperty Name "Channel_2"}
	Channel_2 : Channel_42CA91F7;
	{attribute addProperty Name "Channel_3"}
	Channel_3 : Channel_42CA91F7;
	{attribute addProperty Name "Channel_4"}
	Channel_4 : Channel_42CA91F7;
	{attribute addProperty Name "Channel_5"}
	Channel_5 : Channel_42CA91F7;
	{attribute addProperty Name "Channel_6"}
	Channel_6 : Channel_42CA91F7;
	{attribute addProperty Name "Channel_7"}
	Channel_7 : Channel_42CA91F7;
	{attribute addProperty Name "Channel_8"}
	Channel_8 : Channel_42CA91F7;
	{attribute addProperty Name "Channel_9"}
	Channel_9 : Channel_42CA91F7;
	{attribute addProperty Name "Channel_10"}
	Channel_10 : Channel_42CA91F7;
	{attribute addProperty Name "Channel_11"}
	Channel_11 : Channel_42CA91F7;
	{attribute addProperty Name "Channel_12"}
	Channel_12 : Channel_42CA91F7;
	{attribute addProperty Name "Channel_13"}
	Channel_13 : Channel_42CA91F7;
	{attribute addProperty Name "Channel_14"}
	Channel_14 : Channel_42CA91F7;
	{attribute addProperty Name "Channel_15"}
	Channel_15 : Channel_42CA91F7;
	{attribute addProperty Name "Channel_16"}
	Channel_16 : Channel_42CA91F7;
	{attribute addProperty Name "WcState"}
	WcState : WcState_0B2B16F9;
	{attribute addProperty Name "InfoData"}
	InfoData : InfoData_6F19DB2B;
END_STRUCT
END_TYPE

// ---- DUTs/IO/Boxes/EL2819_3C4AB9A7.TcDUT
{attribute 'GeneratedUsingTerminal: EL2819-0000-0016'}
{attribute addProperty BoxType "EL2819-0000-0016"}
{attribute addProperty Description "EL2819 16Ch. Dig. Output 24V, 0,5A, Diagnostic"}
{attribute addProperty Physics "KK"}
{attribute addProperty Id "DIG_Diag_InputsAT %I*DIG_Diag_Inputs_F289D61564DIG_Inputs_DeviceAT %I*DIG_Inputs_Device_A1F150A94DIG_OutputsAT %Q*DIG_Outputs_B9300CB616WcStateAT %I*WcState_9091E0EB2InfoDataAT %I*InfoData_32EB74EA10"}
{attribute addProperty CRC "1011530151"}
{attribute addProperty Size "96"}
TYPE EL2819_3C4AB9A7 EXTENDS EtcSlaveTerminalBase_947E5A46 :
STRUCT
	{attribute addProperty Name "DIG_Diag_Inputs"}
	DIG_Diag_Inputs : DIG_Diag_Inputs_F289D615;
	{attribute addProperty Name "DIG_Inputs_Device"}
	DIG_Inputs_Device : DIG_Inputs_Device_A1F150A9;
	{attribute addProperty Name "DIG_Outputs"}
	DIG_Outputs : DIG_Outputs_B9300CB6;
	{attribute addProperty Name "WcState"}
	WcState : WcState_9091E0EB;
	{attribute addProperty Name "InfoData"}
	InfoData : InfoData_32EB74EA;
END_STRUCT
END_TYPE

// ---- DUTs/IO/Boxes/EL2828_E2806B95.TcDUT
{attribute 'GeneratedUsingTerminal: EL2828-0000-0016'}
{attribute addProperty BoxType "EL2828-0000-0016"}
{attribute addProperty Description "EL2828 8Ch. Dig. Output 24V, 2A"}
{attribute addProperty Physics "KK"}
{attribute addProperty Id "Channel_1AT %Q*Channel_42CA91F71Channel_2AT %Q*Channel_42CA91F71Channel_3AT %Q*Channel_42CA91F71Channel_4AT %Q*Channel_42CA91F71Channel_5AT %Q*Channel_42CA91F71Channel_6AT %Q*Channel_42CA91F71Channel_7AT %Q*Channel_42CA91F71Channel_8AT %Q*Channel_42CA91F71WcStateAT %I*WcState_0B2B16F91InfoDataAT %I*InfoData_6F19DB2B2"}
{attribute addProperty CRC "3800066965"}
{attribute addProperty Size "11"}
TYPE EL2828_E2806B95 EXTENDS EtcSlaveTerminalBase_947E5A46 :
STRUCT
	{attribute addProperty Name "Channel_1"}
	Channel_1 : Channel_42CA91F7;
	{attribute addProperty Name "Channel_2"}
	Channel_2 : Channel_42CA91F7;
	{attribute addProperty Name "Channel_3"}
	Channel_3 : Channel_42CA91F7;
	{attribute addProperty Name "Channel_4"}
	Channel_4 : Channel_42CA91F7;
	{attribute addProperty Name "Channel_5"}
	Channel_5 : Channel_42CA91F7;
	{attribute addProperty Name "Channel_6"}
	Channel_6 : Channel_42CA91F7;
	{attribute addProperty Name "Channel_7"}
	Channel_7 : Channel_42CA91F7;
	{attribute addProperty Name "Channel_8"}
	Channel_8 : Channel_42CA91F7;
	{attribute addProperty Name "WcState"}
	WcState : WcState_0B2B16F9;
	{attribute addProperty Name "InfoData"}
	InfoData : InfoData_6F19DB2B;
END_STRUCT
END_TYPE

// ---- DUTs/IO/Boxes/EL2872_2B6483BD.TcDUT
{attribute 'GeneratedUsingTerminal: EL2872-0000-0016'}
{attribute addProperty BoxType "EL2872-0000-0016"}
{attribute addProperty Description "EL2872 16Ch. Dig. Output 24V, 0.5A"}
{attribute addProperty Physics "KK"}
{attribute addProperty Id "Channel_1AT %Q*Channel_42CA91F71Channel_2AT %Q*Channel_42CA91F71Channel_3AT %Q*Channel_42CA91F71Channel_4AT %Q*Channel_42CA91F71Channel_5AT %Q*Channel_42CA91F71Channel_6AT %Q*Channel_42CA91F71Channel_7AT %Q*Channel_42CA91F71Channel_8AT %Q*Channel_42CA91F71Channel_9AT %Q*Channel_42CA91F71Channel_10AT %Q*Channel_42CA91F71Channel_11AT %Q*Channel_42CA91F71Channel_12AT %Q*Channel_42CA91F71Channel_13AT %Q*Channel_42CA91F71Channel_14AT %Q*Channel_42CA91F71Channel_15AT %Q*Channel_42CA91F71Channel_16AT %Q*Channel_42CA91F71WcStateAT %I*WcState_0B2B16F91InfoDataAT %I*InfoData_6F19DB2B2"}
{attribute addProperty CRC "728007613"}
{attribute addProperty Size "19"}
TYPE EL2872_2B6483BD EXTENDS EtcSlaveTerminalBase_947E5A46 :
STRUCT
	{attribute addProperty Name "Channel_1"}
	Channel_1 : Channel_42CA91F7;
	{attribute addProperty Name "Channel_2"}
	Channel_2 : Channel_42CA91F7;
	{attribute addProperty Name "Channel_3"}
	Channel_3 : Channel_42CA91F7;
	{attribute addProperty Name "Channel_4"}
	Channel_4 : Channel_42CA91F7;
	{attribute addProperty Name "Channel_5"}
	Channel_5 : Channel_42CA91F7;
	{attribute addProperty Name "Channel_6"}
	Channel_6 : Channel_42CA91F7;
	{attribute addProperty Name "Channel_7"}
	Channel_7 : Channel_42CA91F7;
	{attribute addProperty Name "Channel_8"}
	Channel_8 : Channel_42CA91F7;
	{attribute addProperty Name "Channel_9"}
	Channel_9 : Channel_42CA91F7;
	{attribute addProperty Name "Channel_10"}
	Channel_10 : Channel_42CA91F7;
	{attribute addProperty Name "Channel_11"}
	Channel_11 : Channel_42CA91F7;
	{attribute addProperty Name "Channel_12"}
	Channel_12 : Channel_42CA91F7;
	{attribute addProperty Name "Channel_13"}
	Channel_13 : Channel_42CA91F7;
	{attribute addProperty Name "Channel_14"}
	Channel_14 : Channel_42CA91F7;
	{attribute addProperty Name "Channel_15"}
	Channel_15 : Channel_42CA91F7;
	{attribute addProperty Name "Channel_16"}
	Channel_16 : Channel_42CA91F7;
	{attribute addProperty Name "WcState"}
	WcState : WcState_0B2B16F9;
	{attribute addProperty Name "InfoData"}
	InfoData : InfoData_6F19DB2B;
END_STRUCT
END_TYPE

// ---- DUTs/IO/Boxes/EL2878_76DE585D.TcDUT
{attribute 'GeneratedUsingTerminal: EL2878-0005-0016'}
{attribute addProperty BoxType "EL2878-0005-0016"}
{attribute addProperty Description "EL2878-0005 8Ch. Dig. Output 24V, 0.5A, Diagnostic"}
{attribute addProperty Physics "KK"}
{attribute addProperty Id "DiagnosticAT %I*Diagnostic_A72B1E171Channel_1AT %Q*Channel_42CA91F71Channel_2AT %Q*Channel_42CA91F71Channel_3AT %Q*Channel_42CA91F71Channel_4AT %Q*Channel_42CA91F71Channel_5AT %Q*Channel_42CA91F71Channel_6AT %Q*Channel_42CA91F71Channel_7AT %Q*Channel_42CA91F71Channel_8AT %Q*Channel_42CA91F71WcStateAT %I*WcState_9091E0EB2InfoDataAT %I*InfoData_6F19DB2B2"}
{attribute addProperty CRC "1994283101"}
{attribute addProperty Size "13"}
TYPE EL2878_76DE585D EXTENDS EtcSlaveTerminalBase_947E5A46 :
STRUCT
	{attribute addProperty Name "Diagnostic"}
	Diagnostic : Diagnostic_A72B1E17;
	{attribute addProperty Name "Channel_1"}
	Channel_1 : Channel_42CA91F7;
	{attribute addProperty Name "Channel_2"}
	Channel_2 : Channel_42CA91F7;
	{attribute addProperty Name "Channel_3"}
	Channel_3 : Channel_42CA91F7;
	{attribute addProperty Name "Channel_4"}
	Channel_4 : Channel_42CA91F7;
	{attribute addProperty Name "Channel_5"}
	Channel_5 : Channel_42CA91F7;
	{attribute addProperty Name "Channel_6"}
	Channel_6 : Channel_42CA91F7;
	{attribute addProperty Name "Channel_7"}
	Channel_7 : Channel_42CA91F7;
	{attribute addProperty Name "Channel_8"}
	Channel_8 : Channel_42CA91F7;
	{attribute addProperty Name "WcState"}
	WcState : WcState_9091E0EB;
	{attribute addProperty Name "InfoData"}
	InfoData : InfoData_6F19DB2B;
END_STRUCT
END_TYPE

// ---- DUTs/IO/Boxes/EL2889_2B6483BD.TcDUT
{attribute 'GeneratedUsingTerminal: EL2889-0000-0016'}
{attribute addProperty BoxType "EL2889-0000-0016"}
{attribute addProperty Description "EL2889 16Ch. Dig. Output 24V, 0.5A, negative"}
{attribute addProperty Physics "KK"}
{attribute addProperty Id "Channel_1AT %Q*Channel_42CA91F71Channel_2AT %Q*Channel_42CA91F71Channel_3AT %Q*Channel_42CA91F71Channel_4AT %Q*Channel_42CA91F71Channel_5AT %Q*Channel_42CA91F71Channel_6AT %Q*Channel_42CA91F71Channel_7AT %Q*Channel_42CA91F71Channel_8AT %Q*Channel_42CA91F71Channel_9AT %Q*Channel_42CA91F71Channel_10AT %Q*Channel_42CA91F71Channel_11AT %Q*Channel_42CA91F71Channel_12AT %Q*Channel_42CA91F71Channel_13AT %Q*Channel_42CA91F71Channel_14AT %Q*Channel_42CA91F71Channel_15AT %Q*Channel_42CA91F71Channel_16AT %Q*Channel_42CA91F71WcStateAT %I*WcState_0B2B16F91InfoDataAT %I*InfoData_6F19DB2B2"}
{attribute addProperty CRC "728007613"}
{attribute addProperty Size "19"}
TYPE EL2889_2B6483BD EXTENDS EtcSlaveTerminalBase_947E5A46 :
STRUCT
	{attribute addProperty Name "Channel_1"}
	Channel_1 : Channel_42CA91F7;
	{attribute addProperty Name "Channel_2"}
	Channel_2 : Channel_42CA91F7;
	{attribute addProperty Name "Channel_3"}
	Channel_3 : Channel_42CA91F7;
	{attribute addProperty Name "Channel_4"}
	Channel_4 : Channel_42CA91F7;
	{attribute addProperty Name "Channel_5"}
	Channel_5 : Channel_42CA91F7;
	{attribute addProperty Name "Channel_6"}
	Channel_6 : Channel_42CA91F7;
	{attribute addProperty Name "Channel_7"}
	Channel_7 : Channel_42CA91F7;
	{attribute addProperty Name "Channel_8"}
	Channel_8 : Channel_42CA91F7;
	{attribute addProperty Name "Channel_9"}
	Channel_9 : Channel_42CA91F7;
	{attribute addProperty Name "Channel_10"}
	Channel_10 : Channel_42CA91F7;
	{attribute addProperty Name "Channel_11"}
	Channel_11 : Channel_42CA91F7;
	{attribute addProperty Name "Channel_12"}
	Channel_12 : Channel_42CA91F7;
	{attribute addProperty Name "Channel_13"}
	Channel_13 : Channel_42CA91F7;
	{attribute addProperty Name "Channel_14"}
	Channel_14 : Channel_42CA91F7;
	{attribute addProperty Name "Channel_15"}
	Channel_15 : Channel_42CA91F7;
	{attribute addProperty Name "Channel_16"}
	Channel_16 : Channel_42CA91F7;
	{attribute addProperty Name "WcState"}
	WcState : WcState_0B2B16F9;
	{attribute addProperty Name "InfoData"}
	InfoData : InfoData_6F19DB2B;
END_STRUCT
END_TYPE

// ---- DUTs/IO/Boxes/EL3174_DCC78662.TcDUT
{attribute 'GeneratedUsingTerminal: EL3174-0030-0016'}
{attribute addProperty BoxType "EL3174-0030-0016"}
{attribute addProperty Description "EL3174-0030 4Ch. Ana. Input +/-10V Diff., +/-20mA SingleEnded, 16 Bit, external calibrated"}
{attribute addProperty Physics "KK"}
{attribute addProperty Id "AI_Standard_Channel_1AT %I*AI_Standard_Channel_A8DF64E310AI_Standard_Channel_2AT %I*AI_Standard_Channel_A8DF64E310AI_Standard_Channel_3AT %I*AI_Standard_Channel_A8DF64E310AI_Standard_Channel_4AT %I*AI_Standard_Channel_A8DF64E310WcStateAT %I*WcState_9091E0EB2InfoDataAT %I*InfoData_32EB74EA10"}
{attribute addProperty CRC "3704063586"}
{attribute addProperty Size "52"}
TYPE EL3174_DCC78662 EXTENDS EtcSlaveTerminalBase_947E5A46 :
STRUCT
	{attribute addProperty Name "AI_Standard_Channel_1"}
	AI_Standard_Channel_1 : AI_Standard_Channel_A8DF64E3;
	{attribute addProperty Name "AI_Standard_Channel_2"}
	AI_Standard_Channel_2 : AI_Standard_Channel_A8DF64E3;
	{attribute addProperty Name "AI_Standard_Channel_3"}
	AI_Standard_Channel_3 : AI_Standard_Channel_A8DF64E3;
	{attribute addProperty Name "AI_Standard_Channel_4"}
	AI_Standard_Channel_4 : AI_Standard_Channel_A8DF64E3;
	{attribute addProperty Name "WcState"}
	WcState : WcState_9091E0EB;
	{attribute addProperty Name "InfoData"}
	InfoData : InfoData_32EB74EA;
END_STRUCT
END_TYPE

// ---- DUTs/IO/Boxes/EL3314_C9476E1C.TcDUT
{attribute 'GeneratedUsingTerminal: EL3314-0030-0021'}
{attribute addProperty BoxType "EL3314-0030-0021"}
{attribute addProperty Description "EL3314-0030 4Ch. Ana Input Thermocouple (TC), High Precision, external calibrated"}
{attribute addProperty Physics "KK"}
{attribute addProperty Id "TC_Inputs_Channel_1AT %I*TC_Inputs_Channel_204FE7509TC_Inputs_Channel_2AT %I*TC_Inputs_Channel_204FE7509TC_Inputs_Channel_3AT %I*TC_Inputs_Channel_204FE7509TC_Inputs_Channel_4AT %I*TC_Inputs_Channel_204FE7509WcStateAT %I*WcState_9091E0EB2InfoDataAT %I*InfoData_32EB74EA10"}
{attribute addProperty CRC "3376901660"}
{attribute addProperty Size "48"}
TYPE EL3314_C9476E1C EXTENDS EtcSlaveTerminalBase_947E5A46 :
STRUCT
	{attribute addProperty Name "TC_Inputs_Channel_1"}
	TC_Inputs_Channel_1 : TC_Inputs_Channel_204FE750;
	{attribute addProperty Name "TC_Inputs_Channel_2"}
	TC_Inputs_Channel_2 : TC_Inputs_Channel_204FE750;
	{attribute addProperty Name "TC_Inputs_Channel_3"}
	TC_Inputs_Channel_3 : TC_Inputs_Channel_204FE750;
	{attribute addProperty Name "TC_Inputs_Channel_4"}
	TC_Inputs_Channel_4 : TC_Inputs_Channel_204FE750;
	{attribute addProperty Name "WcState"}
	WcState : WcState_9091E0EB;
	{attribute addProperty Name "InfoData"}
	InfoData : InfoData_32EB74EA;
END_STRUCT
END_TYPE

// ---- DUTs/IO/Boxes/EL3201_F37BFE85.TcDUT
{attribute 'GeneratedUsingTerminal: EL3201-0030-0022'}
{attribute addProperty BoxType "EL3201-0030-0022"}
{attribute addProperty Description "EL3201-0030 1Ch. Ana. Input PT100 (RTD), High Precision, external calibrated"}
{attribute addProperty Physics "KK"}
{attribute addProperty Id "RTDAT %I*AI_Standard_Channel_4A3944819WcStateAT %I*WcState_9091E0EB2InfoDataAT %I*InfoData_32EB74EA10"}
{attribute addProperty CRC "4084989573"}
{attribute addProperty Size "21"}
TYPE EL3201_F37BFE85 EXTENDS EtcSlaveTerminalBase_947E5A46 :
STRUCT
	{attribute addProperty Name "RTD"}
	RTD : AI_Standard_Channel_4A394481;
	{attribute addProperty Name "WcState"}
	WcState : WcState_9091E0EB;
	{attribute addProperty Name "InfoData"}
	InfoData : InfoData_32EB74EA;
END_STRUCT
END_TYPE

// ---- DUTs/IO/Boxes/EL3202_27F12237.TcDUT
{attribute 'GeneratedUsingTerminal: EL3202-0030-0022'}
{attribute addProperty BoxType "EL3202-0030-0022"}
{attribute addProperty Description "EL3202-0030 2Ch. Ana. Input PT100 (RTD), High Precision, external calibrated"}
{attribute addProperty Physics "KK"}
{attribute addProperty Id "RTD_Inputs_Channel_1AT %I*AI_Standard_Channel_4A3944819RTD_Inputs_Channel_2AT %I*AI_Standard_Channel_4A3944819WcStateAT %I*WcState_9091E0EB2InfoDataAT %I*InfoData_32EB74EA10"}
{attribute addProperty CRC "670114359"}
{attribute addProperty Size "30"}
TYPE EL3202_27F12237 EXTENDS EtcSlaveTerminalBase_947E5A46 :
STRUCT
	{attribute addProperty Name "RTD_Inputs_Channel_1"}
	RTD_Inputs_Channel_1 : AI_Standard_Channel_4A394481;
	{attribute addProperty Name "RTD_Inputs_Channel_2"}
	RTD_Inputs_Channel_2 : AI_Standard_Channel_4A394481;
	{attribute addProperty Name "WcState"}
	WcState : WcState_9091E0EB;
	{attribute addProperty Name "InfoData"}
	InfoData : InfoData_32EB74EA;
END_STRUCT
END_TYPE

// ---- DUTs/IO/Boxes/EL3356_1EAAA6FF.TcDUT
{attribute 'GeneratedUsingTerminal: EL3356-0030-0025'}
{attribute addProperty BoxType "EL3356-0030-0025"}
{attribute addProperty Description "EL3356-0030 1Ch. Ana. Input Resistor Bridge Terminal, 24bit, High Precision, external calibrated"}
{attribute addProperty Physics "KK"}
{attribute addProperty Id "RMB_StatusAT %I*RMB_Status_C0E100AA7RMB_Value_INT32AT %I*RMB_Value_INT_E9189C4B4RMB_ControlAT %Q*RMB_Control_CC49845C5WcStateAT %I*WcState_9091E0EB2InfoDataAT %I*InfoData_32EB74EA10"}
{attribute addProperty CRC "514500351"}
{attribute addProperty Size "28"}
TYPE EL3356_1EAAA6FF EXTENDS EtcSlaveTerminalBase_947E5A46 :
STRUCT
	{attribute addProperty Name "RMB_Status"}
	RMB_Status : RMB_Status_C0E100AA;
	{attribute addProperty Name "RMB_Value_INT32"}
	RMB_Value_INT32 : RMB_Value_INT_E9189C4B;
	{attribute addProperty Name "RMB_Control"}
	RMB_Control : RMB_Control_CC49845C;
	{attribute addProperty Name "WcState"}
	WcState : WcState_9091E0EB;
	{attribute addProperty Name "InfoData"}
	InfoData : InfoData_32EB74EA;
END_STRUCT
END_TYPE

// ---- DUTs/IO/Boxes/EL1502_55AAB421.TcDUT
{attribute 'GeneratedUsingTerminal: EL1502--0000'}
{attribute addProperty BoxType "EL1502--0000"}
{attribute addProperty Description "EL1502 2Ch. +/- Counter 24V, 100kHz"}
{attribute addProperty Physics "KK"}
{attribute addProperty Id "CNT_InputsAT %I*CNT_Inputs_7D4495CD11CNT_OutputsAT %Q*CNT_Outputs_EB14A6758WcStateAT %I*WcState_9091E0EB2InfoDataAT %I*InfoData_32EB74EA10"}
{attribute addProperty CRC "1437250593"}
{attribute addProperty Size "31"}
TYPE EL1502_55AAB421 EXTENDS EtcSlaveTerminalBase_947E5A46 :
STRUCT
	{attribute addProperty Name "CNT_Inputs"}
	CNT_Inputs : CNT_Inputs_7D4495CD;
	{attribute addProperty Name "CNT_Outputs"}
	CNT_Outputs : CNT_Outputs_EB14A675;
	{attribute addProperty Name "WcState"}
	WcState : WcState_9091E0EB;
	{attribute addProperty Name "InfoData"}
	InfoData : InfoData_32EB74EA;
END_STRUCT
END_TYPE

// ---- DUTs/IO/Boxes/EL1502_0B55A582.TcDUT
{attribute 'GeneratedUsingTerminal: EL1502-0000-0001'}
{attribute addProperty BoxType "EL1502-0000-0001"}
{attribute addProperty Description "EL1502 2Ch. +/- Counter 24V, 100kHz"}
{attribute addProperty Physics "KK"}
{attribute addProperty Id "CNT_InputsAT %I*CNT_Inputs_147BF88E12CNT_OutputsAT %Q*CNT_Outputs_EB14A6758WcStateAT %I*WcState_9091E0EB2InfoDataAT %I*InfoData_32EB74EA10"}
{attribute addProperty CRC "190162306"}
{attribute addProperty Size "32"}
TYPE EL1502_0B55A582 EXTENDS EtcSlaveTerminalBase_947E5A46 :
STRUCT
	{attribute addProperty Name "CNT_Inputs"}
	CNT_Inputs : CNT_Inputs_147BF88E;
	{attribute addProperty Name "CNT_Outputs"}
	CNT_Outputs : CNT_Outputs_EB14A675;
	{attribute addProperty Name "WcState"}
	WcState : WcState_9091E0EB;
	{attribute addProperty Name "InfoData"}
	InfoData : InfoData_32EB74EA;
END_STRUCT
END_TYPE

// ---- DUTs/IO/Boxes/EL1502_160D2F0C.TcDUT
{attribute 'GeneratedUsingTerminal: EL1502-0000-0018'}
{attribute addProperty BoxType "EL1502-0000-0018"}
{attribute addProperty Description "EL1502 2Ch. +/- Counter 24V, 100kHz"}
{attribute addProperty Physics "KK"}
{attribute addProperty Id "CNT_InputsAT %I*CNT_Inputs_B6C38E7112CNT_OutputsAT %Q*CNT_Outputs_458039AE8WcStateAT %I*WcState_9091E0EB2InfoDataAT %I*InfoData_32EB74EA10"}
{attribute addProperty CRC "369962764"}
{attribute addProperty Size "32"}
TYPE EL1502_160D2F0C EXTENDS EtcSlaveTerminalBase_947E5A46 :
STRUCT
	{attribute addProperty Name "CNT_Inputs"}
	CNT_Inputs : CNT_Inputs_B6C38E71;
	{attribute addProperty Name "CNT_Outputs"}
	CNT_Outputs : CNT_Outputs_458039AE;
	{attribute addProperty Name "WcState"}
	WcState : WcState_9091E0EB;
	{attribute addProperty Name "InfoData"}
	InfoData : InfoData_32EB74EA;
END_STRUCT
END_TYPE

// ---- DUTs/IO/Boxes/EL1512_FBA8C099.TcDUT
{attribute 'GeneratedUsingTerminal: EL1512-0000-0016'}
{attribute addProperty BoxType "EL1512-0000-0016"}
{attribute addProperty Description "EL1512 2Ch. +/- Counter 24V, 1kHz"}
{attribute addProperty Physics "KK"}
{attribute addProperty Id "CNT_Inputs_Channel_1AT %I*CNT_Inputs_Channel_21E1BB398CNT_Inputs_Channel_2AT %I*CNT_Inputs_Channel_21E1BB398CNT_Outputs_Channel_1AT %Q*CNT_Outputs_Channel_774A30BC6CNT_Outputs_Channel_2AT %Q*CNT_Outputs_Channel_774A30BC6WcStateAT %I*WcState_9091E0EB2InfoDataAT %I*InfoData_32EB74EA10"}
{attribute addProperty CRC "4222140569"}
{attribute addProperty Size "40"}
TYPE EL1512_FBA8C099 EXTENDS EtcSlaveTerminalBase_947E5A46 :
STRUCT
	{attribute addProperty Name "CNT_Inputs_Channel_1"}
	CNT_Inputs_Channel_1 : CNT_Inputs_Channel_21E1BB39;
	{attribute addProperty Name "CNT_Inputs_Channel_2"}
	CNT_Inputs_Channel_2 : CNT_Inputs_Channel_21E1BB39;
	{attribute addProperty Name "CNT_Outputs_Channel_1"}
	CNT_Outputs_Channel_1 : CNT_Outputs_Channel_774A30BC;
	{attribute addProperty Name "CNT_Outputs_Channel_2"}
	CNT_Outputs_Channel_2 : CNT_Outputs_Channel_774A30BC;
	{attribute addProperty Name "WcState"}
	WcState : WcState_9091E0EB;
	{attribute addProperty Name "InfoData"}
	InfoData : InfoData_32EB74EA;
END_STRUCT
END_TYPE

